(* CODESYS project Core.library
   Version: 1.3.3
   Title: Core
   DefaultNamespace: Core
   Placeholder: Core
   Company: Beckhoff Automation LLC

Project tree, tasks and I/O mapping:
  libraries: Tc2_Standard, * (Beckhoff Automation GmbH); Tc2_System, * (Beckhoff Automation GmbH); Tc3_DynamicMemory, * (Beckhoff Automation GmbH); Tc3_EventLogger, * (Beckhoff Automation GmbH); Tc3_JsonXml, * (Beckhoff Automation GmbH); Tc3_Module, * (Beckhoff Automation GmbH); Tc3_PackML_V3, * (Beckhoff Automation GmbH)
  _Interface/
    interface I_Base
    interface I_Command: Execute
    interface I_Disposable: Dispose
    interface I_Enablable: Disable, Enable, Enabled
    interface I_Initializable: Initialize, Initialized
    interface I_Override: Override
    interface I_Resettable: Reset
    interface I_Simulatable: Simulated
    interface I_Stoppable: Stop, Stopped
    interface I_TaskResult: Busy, Error, ErrorId
    interface I_ToString: ToString
  _Internal/
    Collection/
      Interface/
        interface I_Collection: AddItem, Clear, Count, IsEmpty, RemoveItem
        interface I_Enumerator: Current, CurrentItem, MoveToNext, ResetIterator
      function block Collection [ST]: FillGaps, AddItem, Clear, Count, Current, CurrentItem, IsEmpty, MoveToNext, RemoveItem, ResetIterator
    CollectionPeeker/
      Interface/
        interface I_CollectionPeeker: CollectionName, FirstItem, LastItem, MoveDownOne, MoveUpOne, PageDown, PageUp, PeekAt, Refresh
        interface I_Peekable: AcceptPeeker
        interface I_Peeker: PeekCollection
      function block CollectionPeeker [ST]: RefreshItems, UpdateEndItem, UpdateFirstItem, CollectionName, FirstItem, Items, LastItem, MoveDownOne, MoveUpOne, PageDown, PageUp, PeekAt, PeekCollection, Refresh
    Component/
      Interface/
        interface I_ComponentCollection: Accept, Count, GetAtIndex, GetComponentByName
        interface I_ContainComponents: Components, DeregisterComponent, DeregisterCyclic, DeregisterInitialize, RegisterComponent, RegisterCyclic, RegisterInitialize
      function block ComponentCollection [ST]: Accept, AddComponent, Count, GetAtIndex, GetComponentByName, RemoveComponent
    Cyclic/
      Interface/
        interface I_Cyclic: CyclicLogic
      function block CyclicRunner [ST]: AddCallee, CallAll, RemoveCallee
    Events/
      function block TcEventClassArguments [ST]: AddString, Clear, Event
    Initialize/
      function block Initializer [ST]: AddInitialize, Initialized, Initializing, RemoveInitialize
    List/
      Interface/
        interface I_List: ContainsItem, GetAtIndex, InsertAtIndex, RemoveAtIndex
      function block List [ST]: AddItem, Clear, RemoveItem, CountListItems, ContainsItem, Count, GetAtIndex, InsertAtIndex, RemoveAtIndex
    Module/
      Interface/
        interface I_ContainModules: DeregisterCyclic, DeregisterInitialize, DeregisterModule, Modules, RegisterCyclic, RegisterInitialize, RegisterModule
        interface I_ModuleCollection: Accept, Count, GetAtIndex, GetModuleByName
      function block ModuleCollection [ST]: Accept, AddModule, Count, GetAtIndex, GetModuleByName, RemoveModule
    Null/
      function block NullComponent [ST]
      function block NullItem [ST]
      function block NullModule [ST]: Accept, Components, DeregisterComponent, DeregisterCyclic, DeregisterInitialize, DeregisterModule, DeregisterWithParent, FB_Init, Modules, Name, RegisterComponent, RegisterCyclic, RegisterInitialize, RegisterModule, RegisterWithParent, ResetComponents, ResetModules
    Statemachine/
      Interface/
        interface I_StateList: AddStateAtIndex, GetStateAtIndex, NumberOfStates
      function block StateList [ST]: AddStateAtIndex, GetStateAtIndex, NumberOfStates
    Tracing/
      Interface/
        interface I_ContainTraceArgument: Arguments
        interface I_ContainTracePublisher: Publisher
        interface I_TraceArgument
        interface I_TraceInstanceLogger: LogMessageInstance
        interface I_TraceLogger: LogMessage
        interface I_TraceMessageInfo: Message, MessageId, Severity
        interface I_TracePublisher: Subscribe, Unsubscribe
        interface I_TraceSourceInfo: SourceId, SourceName, TimeStamp
      function block AdsLogger [ST]: FB_Init, LogMessage
      function block TcEventLogger [ST]: FB_Init, LogMessage
      function block TraceMessageInfo [ST]: Message, MessageId, Severity
      function block TraceSourceInfo [ST]: SourceId, SourceName, TimeStamp
      function USINT_To_TcEventSeverity [ST]
    Types/
      data type RegistrationResult
  Component/
    Interface/
      interface I_Component: Accept, DeregisterWithParent, Name, RegisterWithParent
      interface I_ComponentVisitor: VisitComponent
    function block Component [ST]: Accept, DeregisterWithParent, Name, RegisterWithParent, FB_Init
    function block CyclicComponent [ST]: CyclicLogic, DeregisterWithParent, RegisterWithParent
  Events/
    Interface/
      interface I_EventArguments: AddString, Clear
      interface I_EventClass: Arguments, ClearEventById, IsResettable, RaiseEvent, ResetBySeverity, SetEvent
      interface I_EventClassTcEvents: GenerateTcEvents, GetHighestActiveEventSeverity
      interface I_EventReaction: GetHighestActiveEventReaction, SetEventReactions
      interface I_EventReactionTcEvents: GetHighestActiveEventSeverity
    function block TcEventClass [ST]: Dispose, FB_Exit, ClearEventById, GetHighestActiveEventReaction, GetHighestActiveEventSeverity, IsResettable, RaiseEvent, ResetBySeverity, SetEvent, SetEventReactions, CheckEventId, FindActiveSeverity, GetEventAutoResetInstance, GetEventInstance, GetEventTriggerInstance, SetEventTriggerInstance, Reset, Arguments, CyclicLogic, GenerateTcEvents
  HMI/
    DUT/
      data type ST_HmiFunction
    Interface/
      interface I_Button: Active, Name, Permissive
      interface I_HmiFunction: ControlType, Disable, Enable, Enabled, InstancePath, LinkObject
      interface I_Permissive: OK, Set
      interface I_StringCollection: AddString, Clear, Entries
    function block Button [ST]: Active, Name, Permissive
    function block HmiFunction [ST]: ControlObject, ControlType, CyclicLogic, Disable, Enable, Enabled, InstancePath, LinkObject
  Modes/
    Interface/
      interface I_Mode: ChangeMode, CurrentMode
    function block ModeControl [ST]: ChangeMode, CurrentMode
    function block PackMLModeControl [ST]: ChangeMode, CurrentMode, CyclicLogic, StateMachine
  Module/
    Interface/
      interface I_Module: Accept, DeregisterWithParent, Name, RegisterWithParent, ResetComponents, ResetModules
      interface I_ModuleVisitor: VisitModule
    function block Module [ST]: FB_Init, CyclicLogic, OnCyclicCall, DeregisterComponent, DeregisterCyclic, DeregisterInitialize, DeregisterModule, DeregisterWithParent, Initialize, Initialized, Initializing, RegisterComponent, RegisterCyclic, RegisterInitialize, RegisterModule, RegisterWithParent, ResetComponents, ResetModules, Accept, Components, Modules, Name
  Module PackML/
    function block PackMLModule [ST]: FB_Init, Aborted, Aborting, Clearing, Completed, Completing, Execute, Held, Holding, Idle, Resetting, Starting, Stopped, Stopping, Suspended, Suspending, Unholding, Unsuspending, CyclicLogic, Statemachine, StateSelect
  Permissive Interlock/
    function block PermissiveInterlock [ST]: Check, OK, Set
  Project Information/
    function F_GetCompany [ST]
    function F_GetTitle [ST]
    function F_GetVersion [ST]
  Statemachine/
    DUT/
      data type ST_PackMLStatemachine_HMI
      data type ST_Statemachine_HMI
    Generic/
      function NextMinorStep [ST]
      function NextStep [ST]
      function SetStep [ST]
      function block State [ST]: Executing, FB_Init, Inactive
      function block Statemachine [ST]: Mode, ChangeState, CurrentState, States, CyclicLogic
      function block Statemachine_HMI [ST]: ControlObject, CyclicLogic, FB_Init
    Interface/
      interface I_ContainStatemachine: Statemachine
      interface I_State: Executing, Inactive
      interface I_Statemachine: ChangeState, CurrentState, Mode, States
    PackML/
      function block NextAvailablePackMLCommands [ST]: GetCommands
      function block PackMLStatemachine [ST]: Mode, CallState, ChangeState, CurrentState, States, CyclicLogic
      function block PackMLStatemachine_HMI [ST]: ControlObject, CyclicLogic, FB_Init
      function block PackMLStatemachine_ModuleIntegrated [ST]: Mode, ChangeState, CurrentState, CyclicLogic, StateComplete, States
  Tracing/
    DUT/
      data type TcEventSeverityExt
    Interface/
      interface I_Trace: Critical, Error, Info, Verbose, Warning
    global variables CoreTrace
    function block Trace [ST]: Critical, Error, Info, LogMessage, Subscribe, TraceLevel, Unsubscribe, Verbose, Warning
  Version/
    global variables Global_Version
  Visitors/
    Enable/
      function block CheckComponentsEnabledVisitor [ST]: Check, Enabled, VisitComponent
      function block DisableAllComponentsVisitor [ST]: Disable, Enabled, VisitComponent
      function block EnableAllComponentsVisitor [ST]: Enable, Enabled, VisitComponent
    Events/
      function block GetActiveEventSeverityVisitor [ST]: ActiveEventSeverity, FB_Init, VisitComponent, VisitModule
    HMI/
      function block GetSystemTreeJsonHmiVisitor [ST]: Clear, FB_Init, GetTree, VisitComponent, VisitModule
      function block HmiEnableDisableAllVisitor [ST]: DisableHmi, EnableHmi, VisitComponent, VisitModule
    Override/
      function block SetAllOverrideVisitor [ST]: Set, VisitComponent, VisitModule
    PackML Statemachine/
      function block ChangePackMLStateOnAllSubModulesVisitor [ST]: ChangeState, VisitModule
      function block EventReactorPackMLVisitor [ST]: CyclicLogic, FB_Init, VisitComponent, VisitModule
    Reset/
      function block GetComponentsTaskResultVisitor [ST]: Busy, Error, ErrorId, Update, VisitComponent
      function block ResetAllVisitor [ST]: Busy, Error, ErrorId, Reset, VisitComponent, VisitModule
      function block ResetComponentsVisitor [ST]: Busy, Error, ErrorId, Reset, VisitComponent
      function block ResetModulesVisitor [ST]: Busy, Error, ErrorId, Reset, VisitModule
    Statemachine/
      function block ChangeModeOnAllSubModulesVisitor [ST]: ChangeMode, VisitModule
      function block ChangeStateOnAllSubModulesVisitor [ST]: ChangeState, VisitModule
      function block EventReactorVisitor [ST]: CyclicLogic, FB_Init, VisitComponent, VisitModule
    Stop/
      function block StopAllComponentsVisitor [ST]: Stop, Stopped, VisitComponent
  global variables CoreParameter
  global variables GlobalCore
*)

// _Internal/Types/RegistrationResult
{attribute 'qualified_only'}
{attribute 'strict'}
{attribute 'to_string'}
TYPE RegistrationResult :
(
	Succeeded := 0,
	NullReference := -1,
	TooManyComponents := -2,
	AlreadyAdded := -3,
	CollectionEmpty := -4,
	NotFoundInCollection := -5
);
END_TYPE

// HMI/DUT/ST_HmiFunction
TYPE ST_HmiFunction :
	STRUCT
		Name	   : STRING;
		HmiEnabled : BOOL := TRUE;
	END_STRUCT
END_TYPE

// Statemachine/DUT/ST_PackMLStatemachine_HMI
TYPE ST_PackMLStatemachine_HMI EXTENDS ST_HmiFunction :
	STRUCT
		// Simplified Control
		ResetPermissive : BOOL;
		ResetPressed	: BOOL;
		Resetted		: BOOL;
		StartPermissive : BOOL;
		StartPressed	: BOOL;
		Started			: BOOL;
		StopPermissive	: BOOL;
		StopPressed		: BOOL;
		Stopped			: BOOL;
		// Standard Control
		CurrentMode	 : DINT;
		ModeCommand	 : DINT;
		CurrentState : E_PMLState;
		StateCommand : E_PMLCommand;
		// Next Available Commands
		NextAvailableCommands : ARRAY[0..9] OF E_PMLCommand;
	END_STRUCT
END_TYPE

// Statemachine/DUT/ST_Statemachine_HMI
TYPE ST_Statemachine_HMI EXTENDS ST_HmiFunction :
	STRUCT
		CurrentState	   : DINT;
		CurrentMode		   : DINT;
		StateChangeCommand : DINT;
		ModeChangeCommand  : DINT;
	END_STRUCT
END_TYPE

// Tracing/DUT/TcEventSeverityExt
{attribute 'qualified_only'}
{attribute 'strict'}
{attribute 'to_string'}
TYPE TcEventSeverityExt : (
		Verbose	 := 0,
		Info	 := 1,
		Warning	 := 2,
		Error	 := 3,
		Critical := 4,
		Off		 := 5
	);
END_TYPE

// Tracing/CoreTrace
VAR_GLOBAL
	Trace : Trace<CoreParameter.MaxCountInCollections> := (TraceLevel := CoreParameter.TraceLevel);
	{attribute 'hide'}
	TcEventLogger : TcEventLogger(Trace);
	{attribute 'hide'}
	AdsLogger : AdsLogger(Trace);
END_VAR

// Version/Global_Version
{attribute 'TcGenerated'}
{attribute 'no-analysis'}
{attribute 'linkalways'}
// This function has been automatically generated from the project information.
VAR_GLOBAL CONSTANT
	{attribute 'const_non_replaced'}
	stLibVersion_Core : ST_LibVersion := (iMajor := 1, iMinor := 3, iBuild := 3, iRevision := 0, nFlags := 0, sVersion := '1.3.3');
END_VAR

// CoreParameter
{attribute 'qualified_only'}
VAR_GLOBAL CONSTANT
	MaxCountInCollections : UDINT			   := 50;
	EnableTcEventLogging  : BOOL			   := FALSE;
	EnableAdsLogger		  : BOOL			   := TRUE;
	ClearingTimeout		  : TIME			   := T#2S;
	TraceLevel			  : TcEventSeverityExt := TcEventSeverityExt.Verbose;
END_VAR

// GlobalCore
{attribute 'qualified_only'}
VAR_GLOBAL
	DynamicMemory : FB_DynMem_Manager;
END_VAR

// _Interface/I_Base
INTERFACE I_Base EXTENDS __SYSTEM.IQueryInterface

END_INTERFACE

// _Interface/I_Command
INTERFACE I_Command EXTENDS I_Base

METHOD Execute : BOOL
VAR_INPUT
END_VAR
END_METHOD

END_INTERFACE

// _Interface/I_Disposable
INTERFACE I_Disposable EXTENDS I_Base

METHOD Dispose
VAR_INPUT
END_VAR
END_METHOD

END_INTERFACE

// _Interface/I_Enablable
INTERFACE I_Enablable EXTENDS I_Base

METHOD Disable
VAR_INPUT
END_VAR
END_METHOD

METHOD Enable
VAR_INPUT
END_VAR
END_METHOD

{attribute 'monitoring' := 'call'}
PROPERTY Enabled : BOOL
GET
END_GET
END_PROPERTY

END_INTERFACE

// _Interface/I_Initializable
INTERFACE I_Initializable EXTENDS I_Base

METHOD Initialize
END_METHOD

{attribute 'monitoring' := 'call'}
PROPERTY Initialized : BOOL
GET
END_GET
SET
END_SET
END_PROPERTY

END_INTERFACE

// _Interface/I_Override
INTERFACE I_Override EXTENDS I_Base

{attribute 'monitoring' := 'call'}
PROPERTY Override : LREAL
SET
END_SET
END_PROPERTY

END_INTERFACE

// _Interface/I_Resettable
INTERFACE I_Resettable EXTENDS I_Base

METHOD Reset
END_METHOD

END_INTERFACE

// _Interface/I_Simulatable
INTERFACE I_Simulatable EXTENDS I_Base

{attribute 'monitoring' := 'call'}
PROPERTY Simulated : BOOL
GET
END_GET
SET
END_SET
END_PROPERTY

END_INTERFACE

// _Interface/I_Stoppable
INTERFACE I_Stoppable EXTENDS I_Base

METHOD Stop
VAR_INPUT
END_VAR
END_METHOD

{attribute 'monitoring' := 'call'}
PROPERTY Stopped : BOOL
GET
END_GET
END_PROPERTY

END_INTERFACE

// _Interface/I_TaskResult
INTERFACE I_TaskResult EXTENDS I_Base

{attribute 'monitoring' := 'call'}
PROPERTY Busy : BOOL
GET
END_GET
END_PROPERTY

{attribute 'monitoring' := 'call'}
PROPERTY Error : BOOL
GET
END_GET
END_PROPERTY

{attribute 'monitoring' := 'call'}
PROPERTY ErrorId : UDINT
GET
END_GET
END_PROPERTY

END_INTERFACE

// _Interface/I_ToString
INTERFACE I_ToString EXTENDS I_Base

METHOD ToString : T_MaxString
VAR_INPUT
END_VAR
END_METHOD

END_INTERFACE

// _Internal/Collection/Interface/I_Collection
INTERFACE I_Collection EXTENDS I_Enumerator

METHOD AddItem
VAR_INPUT
	Item : I_Base;
END_VAR
END_METHOD

METHOD Clear
VAR_INPUT
END_VAR
END_METHOD

{attribute 'monitoring' := 'call'}
PROPERTY Count : UDINT
GET
END_GET
END_PROPERTY

{attribute 'monitoring' := 'call'}
PROPERTY IsEmpty : BOOL
GET
END_GET
END_PROPERTY

METHOD RemoveItem
VAR_INPUT
	Item : I_Base;
END_VAR
END_METHOD

END_INTERFACE

// _Internal/Collection/Interface/I_Enumerator
INTERFACE I_Enumerator

PROPERTY Current : I_Base
GET
END_GET
END_PROPERTY

{attribute 'monitoring' := 'call'}
PROPERTY CurrentItem : UDINT
GET
END_GET
END_PROPERTY

PROPERTY MoveToNext : BOOL
GET
END_GET
END_PROPERTY

METHOD ResetIterator
VAR_INPUT
END_VAR
END_METHOD

END_INTERFACE

// _Internal/Collection/Collection
FUNCTION_BLOCK Collection
VAR_GENERIC CONSTANT
	CollectionSize : UDINT := 1;
END_VAR IMPLEMENTS I_Collection, I_Enumerator
VAR
	{attribute 'instance-path'}
	{attribute 'noinit'}
	InstancePath  : STRING;
	_Data		  : ARRAY[0..CollectionSize - 1] OF I_Base;
	_Current	  : I_Base;
	_Count		  : UDINT;
	_CurrentIndex : UDINT;
	{attribute 'hide'}
	NullItem : NullItem;
	{attribute 'hide'}
	ipNullItem : I_Base := NullItem;
END_VAR

METHOD PROTECTED FillGaps
VAR
	Item	 : I_Base;
	ItemNext : I_Base;
	i		 : UDINT;
END_VAR
IF _Count > 1 THEN
	FOR i := 0 TO (_Count - 2) DO
		Item	 := _Data[i];
		ItemNext := _Data[i + 1];
		IF Item = 0 AND ItemNext <> 0 THEN
			_Data[i]	 := ItemNext;
			_Data[i + 1] := 0;
		END_IF
	END_FOR
END_IF
END_METHOD

METHOD AddItem
VAR_INPUT
	Item	: I_Base;
END_VAR
IF Item = 0 THEN
	Trace.Error(InstancePath, 'No Items to add to this Collection!');
	RETURN;
END_IF

IF _Count > CollectionSize - 1 THEN
	Trace.Error(InstancePath, 'No space left in Collection, increase size!');
	RETURN;
END_IF

_Data[_Count] := Item;
_Count		  := _Count + 1;
END_METHOD

METHOD Clear
VAR
	i : UDINT;
END_VAR
IF _Count = 0 THEN
	RETURN;
END_IF

FOR i := 0 TO _Count - 1 DO
	_Data[i] := 0;
END_FOR

_Count := 0;
ResetIterator();
END_METHOD

{attribute 'monitoring' := 'call'}
PROPERTY Count : UDINT
GET
Count := _Count;
END_GET
END_PROPERTY

PROPERTY Current : I_Base
GET
IF _Current <> 0 THEN
	Current := _Current; 
END_IF
END_GET
END_PROPERTY

{attribute 'monitoring' := 'call'}
PROPERTY CurrentItem : UDINT
GET
CurrentItem := _CurrentIndex;
END_GET
END_PROPERTY

{attribute 'monitoring' := 'call'}
PROPERTY IsEmpty : BOOL
GET
IsEmpty := _Count = 0;
END_GET
END_PROPERTY

PROPERTY MoveToNext : BOOL
GET
MoveToNext := FALSE;
IF Count = 0 THEN
	RETURN;
END_IF

IF _CurrentIndex = Count THEN
	RETURN;
END_IF

_Current	  := _Data[_CurrentIndex];
_CurrentIndex := _CurrentIndex + 1;
MoveToNext	  := TRUE;
END_GET
END_PROPERTY

METHOD RemoveItem
VAR_INPUT
	Item : I_Base;
END_VAR

VAR
	i		  : UDINT;
	ItemFound : BOOL;
END_VAR
IF _Count = 0 THEN
	Trace.LogMessage(InstancePath, 'No Items found in this Collection!');
	RETURN;
END_IF

IF Item = 0 THEN
	Trace.LogMessage(InstancePath, 'Item to remove needs to be valid interface!');
	RETURN;
END_IF

FOR i := 0 TO (_Count - 1) DO
	IF _Data[i] = Item THEN
		_Data[i]  := 0;
		ItemFound := TRUE;
	END_IF
END_FOR

FillGaps();
IF ItemFound THEN
	_Count := _Count - 1;
END_IF
END_METHOD

METHOD ResetIterator
_Current	  := ipNullItem;
_CurrentIndex := 0;
END_METHOD

END_FUNCTION_BLOCK

// _Internal/Null/NullItem
FUNCTION_BLOCK NullItem IMPLEMENTS I_Base
VAR
END_VAR

END_FUNCTION_BLOCK

// Tracing/Trace
FUNCTION_BLOCK Trace
VAR_GENERIC CONSTANT
	MaxCount : UDINT := 10;
END_VAR IMPLEMENTS I_TracePublisher, I_Trace
VAR
	Loggers : ARRAY[0..MaxCount] OF I_TraceLogger;
	_TraceLevel : TcEventSeverityExt := TcEventSeverityExt.Warning;
END_VAR

METHOD Critical
VAR_INPUT
	Source	  : T_MaxString;
	Message	  : T_MaxString;
END_VAR
VAR
	i : UDINT;
END_VAR
FOR i := 0 TO MaxCount DO
	IF Loggers[i] <> 0 AND_THEN _TraceLevel < 5 THEN
		Loggers[i].LogMessage(Source,
							  Message,
							  0,
							  0,
							  1,
							  4);
	END_IF
END_FOR
END_METHOD

METHOD Error
VAR_INPUT
	Source	  : T_MaxString;
	Message	  : T_MaxString;
END_VAR
VAR
	i : UDINT;
END_VAR
FOR i := 0 TO MaxCount DO
	IF Loggers[i] <> 0 AND_THEN _TraceLevel < 4 THEN
		Loggers[i].LogMessage(Source,
							  Message,
							  0,
							  0,
							  1,
							  3);
	END_IF
END_FOR
END_METHOD

METHOD Info
VAR_INPUT
	Source	  : T_MaxString;
	Message	  : T_MaxString;
END_VAR
VAR
	i : UDINT;
END_VAR
FOR i := 0 TO MaxCount DO
	IF Loggers[i] <> 0 AND_THEN _TraceLevel < 2 THEN
		Loggers[i].LogMessage(Source,
							  Message,
							  0,
							  0,
							  1,
							  1);
	END_IF
END_FOR
END_METHOD

METHOD LogMessage
VAR_INPUT
	Key		  : T_MaxString;
	Value	  : T_MaxString;
	SourceId  : UDINT := 0;
	TimeStamp : ULINT := 0;
	MessageId : UDINT := 1;
	Severity  : USINT := 1;
END_VAR

VAR
	i : UDINT;
END_VAR
FOR i := 0 TO MaxCount DO
	IF Loggers[i] <> 0 THEN
		Loggers[i].LogMessage(Key,
							  Value,
							  SourceId,
							  TimeStamp,
							  MessageId,
							  Severity);
	END_IF
END_FOR
END_METHOD

METHOD Subscribe
VAR_INPUT
	Logger : I_TraceLogger;
END_VAR

VAR
	i : UDINT;
END_VAR
FOR i := 0 TO CoreParameter.MaxCountInCollections DO
	IF Loggers[i] = 0 THEN
		Loggers[i] := Logger;
		EXIT;
	END_IF
END_FOR
END_METHOD

PROPERTY TraceLevel : TcEventSeverityExt
GET
TraceLevel := _TraceLevel;
END_GET
SET
_TraceLevel := TraceLevel;
END_SET
END_PROPERTY

METHOD Unsubscribe
VAR_INPUT
	Logger : I_TraceLogger;
END_VAR

VAR
	i : UDINT;
END_VAR
FOR i := 0 TO CoreParameter.MaxCountInCollections DO
	IF Loggers[i] = Logger THEN
		Loggers[i] := 0;
		EXIT;
	END_IF
END_FOR
END_METHOD

METHOD Verbose
VAR_INPUT
	Source	  : T_MaxString;
	Message	  : T_MaxString;
END_VAR
VAR
	i : UDINT;
END_VAR
FOR i := 0 TO MaxCount DO
	IF Loggers[i] <> 0 AND_THEN _TraceLevel = 0 THEN
		Loggers[i].LogMessage(Source,
							  Message,
							  0,
							  0,
							  1,
							  0);
	END_IF
END_FOR
END_METHOD

METHOD Warning
VAR_INPUT
	Source	  : T_MaxString;
	Message	  : T_MaxString;
END_VAR
VAR
	i : UDINT;
END_VAR
FOR i := 0 TO MaxCount DO
	IF Loggers[i] <> 0 AND_THEN _TraceLevel < 3 THEN
		Loggers[i].LogMessage(Source,
							  Message,
							  0,
							  0,
							  1,
							  2);
	END_IF
END_FOR
END_METHOD

END_FUNCTION_BLOCK

// _Internal/Tracing/Interface/I_TracePublisher
INTERFACE I_TracePublisher

METHOD Subscribe
VAR_INPUT
	Logger : I_TraceLogger;
END_VAR
END_METHOD

METHOD Unsubscribe
VAR_INPUT
	Logger : I_TraceLogger;
END_VAR
END_METHOD

END_INTERFACE

// _Internal/Tracing/Interface/I_TraceLogger
INTERFACE I_TraceLogger EXTENDS I_Base

METHOD LogMessage
VAR_INPUT
	Key		  : T_MaxString;
	Value	  : T_MaxString;
	SourceId  : UDINT := 0;
	TimeStamp : ULINT := 0;
	MessageId : UDINT := 1;
	Severity  : USINT := 1;
END_VAR
END_METHOD

END_INTERFACE

// Tracing/Interface/I_Trace
INTERFACE I_Trace

METHOD Critical
VAR_INPUT
	Source	  : T_MaxString;
	Message	  : T_MaxString;
END_VAR
END_METHOD

METHOD Error
VAR_INPUT
	Source	  : T_MaxString;
	Message	  : T_MaxString;
END_VAR
END_METHOD

METHOD Info
VAR_INPUT
	Source	  : T_MaxString;
	Message	  : T_MaxString;
END_VAR
END_METHOD

METHOD Verbose
VAR_INPUT
	Source	  : T_MaxString;
	Message	  : T_MaxString;
END_VAR
END_METHOD

METHOD Warning
VAR_INPUT
	Source	  : T_MaxString;
	Message	  : T_MaxString;
END_VAR
END_METHOD

END_INTERFACE

// _Internal/CollectionPeeker/Interface/I_CollectionPeeker
INTERFACE I_CollectionPeeker EXTENDS I_Base

{attribute 'monitoring':='call'}
PROPERTY CollectionName : T_MaxString
GET
END_GET
SET
END_SET
END_PROPERTY

{attribute 'monitoring':='call'}
PROPERTY FirstItem : UDINT
GET
END_GET
END_PROPERTY

{attribute 'monitoring':='call'}
PROPERTY LastItem : UDINT
GET
END_GET
END_PROPERTY

{attribute 'monitoring' := 'call'}
PROPERTY MoveDownOne : BOOL
SET
END_SET
END_PROPERTY

{attribute 'monitoring' := 'call'}
PROPERTY MoveUpOne : BOOL
SET
END_SET
END_PROPERTY

{attribute 'monitoring' := 'call'}
PROPERTY PageDown : BOOL
SET
END_SET
END_PROPERTY

{attribute 'monitoring' := 'call'}
PROPERTY PageUp : BOOL
SET
END_SET
END_PROPERTY

METHOD PeekAt
VAR_INPUT
	Peekable : I_Peekable;
END_VAR
END_METHOD

{attribute 'monitoring':='call'}
PROPERTY Refresh : BOOL
GET
END_GET
SET
END_SET
END_PROPERTY

END_INTERFACE

// _Internal/CollectionPeeker/Interface/I_Peekable
INTERFACE I_Peekable EXTENDS I_Base

METHOD AcceptPeeker
VAR_INPUT
	Peeker : I_Peeker;
END_VAR
END_METHOD

END_INTERFACE

// _Internal/CollectionPeeker/Interface/I_Peeker
INTERFACE I_Peeker EXTENDS I_Base

METHOD PeekCollection
VAR_INPUT
	Collection : I_Collection;
END_VAR
END_METHOD

END_INTERFACE

// _Internal/CollectionPeeker/CollectionPeeker
{attribute 'hide_all_locals'}
FUNCTION_BLOCK CollectionPeeker
VAR_GENERIC CONSTANT
	Peek_Size : UDINT := 5;
END_VAR IMPLEMENTS I_CollectionPeeker, I_Peeker
VAR
	_CurrentItem	: UDINT;
	_EndItem		: UDINT;
	_CollectionName : T_MaxString;
	_Collection		: I_Collection;
	_Items			: ARRAY[1..Peek_Size] OF I_Base;
END_VAR

METHOD PRIVATE RefreshItems
VAR
	startItem  : UDINT;
	endItem	   : UDINT;
	i		   : UDINT := 1;
	wrapAround : BOOL;
END_VAR
MEMSET(ADR(_Items), 0, SIZEOF(_Items));
IF _CurrentItem > _EndItem THEN //we're wrapped around
	i		   := 1 + ((_Collection.Count - _CurrentItem) + 1);
	wrapAround := TRUE;
END_IF

_Collection.ResetIterator();
WHILE _Collection.MoveToNext DO
	IF _Collection.CurrentItem >= _CurrentItem AND _Collection.CurrentItem <= _EndItem THEN
		_Items[i] := _Collection.Current;
		i		  := i + 1;
	ELSIF wrapAround AND (_Collection.CurrentItem >= _CurrentItem OR _Collection.CurrentItem <= _EndItem) THEN
		_Items[i] := _Collection.Current;
		i		  := i + 1;
		IF i > Peek_Size THEN
			i := 1;
		END_IF
	END_IF
END_WHILE
END_METHOD

METHOD PRIVATE UpdateEndItem
VAR_INPUT
END_VAR
_EndItem := _CurrentItem + Peek_Size - 1;
IF _EndItem > _Collection.Count THEN
	_EndItem := _EndItem - _Collection.Count;
END_IF
END_METHOD

METHOD PRIVATE UpdateFirstItem
VAR_INPUT
END_VAR
END_METHOD

{attribute 'monitoring':='call'}
PROPERTY CollectionName : T_MaxString
GET
CollectionName := _CollectionName;
END_GET
SET
_CollectionName := CollectionName;
END_SET
END_PROPERTY

{attribute 'monitoring' := 'call'}
PROPERTY FirstItem : UDINT
GET
FirstItem := _CurrentItem;
END_GET
SET
IF _Collection = 0 THEN
	RETURN;
END_IF

IF FirstItem > _Collection.Count OR FirstItem < 1 THEN
	RETURN;
END_IF

_CurrentItem := FirstItem;
UpdateEndItem();
RefreshItems();
END_SET
END_PROPERTY

{attribute 'monitoring' := 'call'}
PROPERTY Items : REFERENCE TO ARRAY[1..Peek_Size] OF I_Base
GET
Items REF= _Items;
END_GET
END_PROPERTY

{attribute 'monitoring' := 'call'}
PROPERTY LastItem : UDINT
GET
LastItem := _EndItem;
END_GET
END_PROPERTY

{attribute 'monitoring' := 'call'}
PROPERTY MoveDownOne : BOOL
GET
END_GET
SET
IF _Collection = 0 OR NOT MoveDownOne THEN
	RETURN;
END_IF

IF _Collection.Count <= Peek_Size THEN
	RETURN;
END_IF

_CurrentItem := _CurrentItem + 1;
IF _CurrentItem > _Collection.Count THEN
	_CurrentItem := 1;
END_IF

UpdateEndItem();
RefreshItems();
END_SET
END_PROPERTY

{attribute 'monitoring' := 'call'}
PROPERTY MoveUpOne : BOOL
GET
END_GET
SET
IF _Collection = 0 THEN
	RETURN;
END_IF

IF _Collection.Count <= Peek_Size THEN
	RETURN;
END_IF

_CurrentItem := _CurrentItem - 1;
IF _CurrentItem < 1 THEN
	_CurrentItem := _Collection.Count;
END_IF

UpdateEndItem();
RefreshItems();
END_SET
END_PROPERTY

{attribute 'monitoring' := 'call'}
PROPERTY PageDown : BOOL
GET
END_GET
SET
IF _Collection = 0 OR NOT PageDown THEN
	RETURN;
END_IF

IF _Collection.Count <= Peek_Size THEN
	RETURN;
END_IF

IF _CurrentItem > (_Collection.Count - Peek_Size) THEN
	_CurrentItem := (Peek_Size - (_Collection.Count - _CurrentItem));
ELSE
	_CurrentItem := _CurrentItem + Peek_Size;
END_IF

UpdateEndItem();
RefreshItems();
END_SET
END_PROPERTY

{attribute 'monitoring' := 'call'}
PROPERTY PageUp : BOOL
GET
END_GET
SET
VAR
	tmp : UDINT;
END_VAR
IF _Collection = 0 OR NOT PageUp THEN
	RETURN;
END_IF

IF _Collection.Count <= Peek_Size THEN
	RETURN;
END_IF

IF _CurrentItem < Peek_Size THEN
	_CurrentItem := (_Collection.Count - (Peek_Size - _CurrentItem));
ELSE
	_CurrentItem := _CurrentItem - Peek_Size;
END_IF

UpdateEndItem();
RefreshItems();
END_SET
END_PROPERTY

METHOD PeekAt
VAR_INPUT
	Peekable : I_Peekable;
END_VAR
Peekable.AcceptPeeker(THIS^);
END_METHOD

METHOD PeekCollection
VAR_INPUT
	Collection : I_Collection;
END_VAR
_Collection	 := Collection;
_CurrentItem := 1;
_EndItem	 := Peek_Size;
RefreshItems();
END_METHOD

{attribute 'monitoring':='call'}
PROPERTY Refresh : BOOL
GET
END_GET
SET
IF _Collection <> 0 AND Refresh THEN
	RefreshItems();
END_IF
END_SET
END_PROPERTY

END_FUNCTION_BLOCK

// _Internal/Component/Interface/I_ComponentCollection
INTERFACE I_ComponentCollection

METHOD Accept
VAR_INPUT
	Visitor : I_ComponentVisitor;
END_VAR
END_METHOD

{attribute 'monitoring' := 'call'}
PROPERTY Count : UDINT
GET
END_GET
END_PROPERTY

METHOD GetAtIndex : I_Component
VAR_INPUT
	Index : UDINT;
END_VAR
END_METHOD

METHOD GetComponentByName : I_Component
VAR_INPUT
	Name : T_MaxString;
END_VAR
END_METHOD

END_INTERFACE

// Component/Interface/I_ComponentVisitor
INTERFACE I_ComponentVisitor

METHOD VisitComponent
VAR_INPUT
	Component : I_Component;
END_VAR
END_METHOD

END_INTERFACE

// Component/Component
FUNCTION_BLOCK ABSTRACT Component IMPLEMENTS I_Component
VAR
	_Name : T_MaxString;
	RegisteredAsComponentResult : RegistrationResult;
END_VAR

METHOD Accept
VAR_INPUT
	ComponentVisitor : I_ComponentVisitor;
END_VAR
ComponentVisitor.VisitComponent(THIS^);
END_METHOD

METHOD DeregisterWithParent
VAR_INPUT
	Parent : I_ContainComponents;
END_VAR
Parent.DeregisterComponent(THIS^);
END_METHOD

{attribute 'monitoring' := 'call'}
PROPERTY Name : T_MaxString
GET
Name := _Name;
END_GET
SET
_Name := Name;
END_SET
END_PROPERTY

METHOD RegisterWithParent
VAR_INPUT
	Parent : I_ContainComponents;
END_VAR
RegisteredAsComponentResult := Parent.RegisterComponent(THIS^);
END_METHOD

//FB_Init is always available implicitly and it is used primarily for initialization.

//The return value is not evaluated. For a specific influence, you can also declare the

//methods explicitly and provide additional code there with the standard initialization

//code. You can evaluate the return value.
METHOD FB_Init : BOOL
VAR_INPUT
	bInitRetains : BOOL; // TRUE: the retain variables are initialized (reset warm / reset cold)
	bInCopyCode	 : BOOL; // TRUE: the instance will be copied to the copy code afterward (online change)   
	Name		 : T_MaxString;
END_VAR
_Name := Name;
END_METHOD

END_FUNCTION_BLOCK

// Component/Interface/I_Component
INTERFACE I_Component EXTENDS I_Base

METHOD Accept
VAR_INPUT
	ComponentVisitor : I_ComponentVisitor;
END_VAR
END_METHOD

METHOD DeregisterWithParent
VAR_INPUT
	Parent : I_ContainComponents;
END_VAR
END_METHOD

{attribute 'monitoring' := 'call'}
PROPERTY Name : T_MaxString
GET
END_GET
SET
END_SET
END_PROPERTY

METHOD RegisterWithParent
VAR_INPUT
	Parent : I_ContainComponents;
END_VAR
END_METHOD

END_INTERFACE

// _Internal/Component/Interface/I_ContainComponents
INTERFACE I_ContainComponents

PROPERTY Components : I_ComponentCollection
GET
END_GET
END_PROPERTY

METHOD DeregisterComponent  : RegistrationResult
VAR_INPUT
	Component : I_Component;
END_VAR
END_METHOD

METHOD DeregisterCyclic : RegistrationResult
VAR_INPUT
	Cyclic : I_Cyclic;
END_VAR
END_METHOD

METHOD DeregisterInitialize : RegistrationResult
VAR_INPUT
	Initializable : I_Initializable;
END_VAR
END_METHOD

METHOD RegisterComponent  : RegistrationResult
VAR_INPUT
	Component : I_Component;
END_VAR
END_METHOD

METHOD RegisterCyclic  : RegistrationResult
VAR_INPUT
	Cyclic : I_Cyclic;
END_VAR
END_METHOD

METHOD RegisterInitialize  : RegistrationResult
VAR_INPUT
	Initializable : I_Initializable;
END_VAR
END_METHOD

END_INTERFACE

// _Internal/Cyclic/Interface/I_Cyclic
INTERFACE I_Cyclic EXTENDS I_Base

METHOD CyclicLogic
VAR_INPUT
END_VAR
END_METHOD

END_INTERFACE

// _Internal/Component/ComponentCollection
FUNCTION_BLOCK ComponentCollection
VAR_GENERIC CONSTANT
	MaxCount : UDINT := 10;
END_VAR IMPLEMENTS I_ComponentCollection
VAR
	Components	   : ARRAY[0..MaxCount] OF I_Component;
	ComponentCount : UDINT;
	NullComponent  : NullComponent('Null Component');
END_VAR

METHOD Accept
VAR_INPUT
	Visitor : I_ComponentVisitor;
END_VAR

VAR
	i : UDINT;
END_VAR
FOR i := 0 TO MaxCount DO
	IF Components[i] = 0 THEN
		EXIT;
	END_IF

	Components[i].Accept(Visitor);
END_FOR
END_METHOD

METHOD AddComponent : RegistrationResult
VAR_INPUT
	Component : I_Component;
END_VAR

VAR
	i : UDINT;
	Registered : BOOL;
END_VAR
IF Component = 0 THEN
	AddComponent := RegistrationResult.NullReference;
	RETURN;
END_IF

IF ComponentCount >= MaxCount THEN
	AddComponent := RegistrationResult.TooManyComponents;
	RETURN;
END_IF

FOR i := 0 TO MaxCount DO
	IF Components[i] = Component THEN
		Registered := TRUE;
	END_IF
END_FOR

IF Registered THEN
	AddComponent := RegistrationResult.AlreadyAdded;
	RETURN;
END_IF

FOR i := 0 TO MaxCount DO
	IF Components[i] = 0 THEN
		Components[i] := Component;
		ComponentCount := ComponentCount + 1;
		EXIT;
	END_IF
END_FOR
END_METHOD

{attribute 'monitoring' := 'call'}
PROPERTY Count : UDINT
GET
Count := TO_UDINT(ComponentCount);
END_GET
END_PROPERTY

METHOD GetAtIndex : I_Component
VAR_INPUT
	Index : UDINT;
END_VAR
IF Index > Count THEN
	GetAtIndex := NullComponent;
	RETURN;
END_IF

IF Index < 0 THEN
	GetAtIndex := NullComponent;
	RETURN;
END_IF

IF Components[Index] <> 0 THEN
	GetAtIndex := Components[Index];
ELSE
	GetAtIndex := NullComponent;
END_IF
END_METHOD

METHOD GetComponentByName : I_Component
VAR_INPUT
	Name : T_MaxString;
END_VAR

VAR
	i : UDINT;
END_VAR
FOR i := 0 TO MaxCount DO
	IF Components[i] = 0 THEN
		EXIT;
	END_IF

	IF Components[i].Name = Name THEN
		GetComponentByName := Components[i];
		EXIT;
	END_IF
END_FOR
END_METHOD

METHOD RemoveComponent : RegistrationResult
VAR_INPUT
	Component : I_Component;
END_VAR

VAR
	i : UDINT;
	PresentInCollection : BOOL;
END_VAR
IF Component = 0 THEN
	RemoveComponent := RegistrationResult.NullReference;
	RETURN;
END_IF

IF ComponentCount = 0 THEN
	RemoveComponent := RegistrationResult.CollectionEmpty;
	RETURN;
END_IF

FOR i := 0 TO MaxCount DO
	IF Components[i] = Component THEN
		PresentInCollection := TRUE;
	END_IF
END_FOR

IF NOT PresentInCollection THEN
	RemoveComponent := RegistrationResult.NotFoundInCollection;
	RETURN;
END_IF

FOR i := 0 TO MaxCount DO
	IF Components[i] = Component THEN
		ComponentCount := ComponentCount - 1;
		IF i < MaxCount THEN
			MEMMOVE(ADR(Components[i]), ADR(Components[i + 1]), (MaxCount - i) * SIZEOF(Component));
		ELSE
			Components[MaxCount] := 0;
		END_IF
		EXIT;
	END_IF
END_FOR
END_METHOD

END_FUNCTION_BLOCK

// _Internal/Null/NullComponent
FUNCTION_BLOCK NullComponent EXTENDS Component
VAR
END_VAR

END_FUNCTION_BLOCK

// _Internal/Cyclic/CyclicRunner
FUNCTION_BLOCK CyclicRunner
VAR_GENERIC CONSTANT
	MaxCount : UDINT := 10;
END_VAR

VAR
	Callees		: ARRAY[0..MaxCount] OF I_Cyclic;
	CalleeCount : UDINT;
END_VAR

METHOD AddCallee : RegistrationResult
VAR_INPUT
	Callee : I_Cyclic;
END_VAR

VAR
	i : UDINT;
	Registered : BOOL;
END_VAR
IF Callee = 0 THEN
	AddCallee := RegistrationResult.NullReference;
	RETURN;
END_IF

IF CalleeCount >= MaxCount THEN
	AddCallee := RegistrationResult.TooManyComponents;
	RETURN;
END_IF

FOR i := 0 TO MaxCount DO
	IF Callees[i] = Callee THEN
		Registered := TRUE;
	END_IF
END_FOR

IF Registered THEN
	AddCallee := RegistrationResult.AlreadyAdded;
	RETURN;
END_IF

FOR i := 0 TO MaxCount DO
	IF Callees[i] = 0 THEN
		Callees[i] := Callee;
		CalleeCount := CalleeCount + 1;
		EXIT;
	END_IF
END_FOR
END_METHOD

METHOD CallAll
VAR_INST
	Logged : BOOL;
END_VAR

VAR
	i	   : UDINT;
	Callee : I_Cyclic;
END_VAR
FOR i := 0 TO MaxCount DO
	IF Callees[i] = 0 THEN
		RETURN;
	END_IF

	Callees[i].CyclicLogic();
END_FOR

IF NOT Logged THEN
	Logged := TRUE;
	Trace.LogMessage('Cyclic Runner', 'Collection is full. Review library parameters and code to ensure proper setup.');
END_IF
END_METHOD

METHOD RemoveCallee : RegistrationResult
VAR_INPUT
	Callee : I_Cyclic;
END_VAR

VAR
	i : UDINT;
	PresentInCollection : BOOL;
END_VAR
IF Callee = 0 THEN
	RemoveCallee := RegistrationResult.NullReference;
	RETURN;
END_IF

IF CalleeCount = 0 THEN
	RemoveCallee := RegistrationResult.CollectionEmpty;
	RETURN;
END_IF

FOR i := 0 TO MaxCount DO
	IF Callees[i] = Callee THEN
		PresentInCollection := TRUE;
	END_IF
END_FOR

IF NOT PresentInCollection THEN
	RemoveCallee := RegistrationResult.NotFoundInCollection;
	RETURN;
END_IF

FOR i := 0 TO MaxCount DO
	IF Callees[i] = Callee THEN
		CalleeCount := CalleeCount - 1;
		IF i < MaxCount THEN
			MEMMOVE(ADR(Callees[i]), ADR(Callees[i + 1]), (MaxCount - i) * SIZEOF(Callee));
		ELSE
			Callees[MaxCount] := 0;
		END_IF
		EXIT;
	END_IF
END_FOR
END_METHOD

END_FUNCTION_BLOCK

// _Internal/Events/TcEventClassArguments
FUNCTION_BLOCK TcEventClassArguments IMPLEMENTS I_EventArguments
VAR
	pArgumentEvent : POINTER TO FB_TcAlarm;
END_VAR

METHOD AddString : I_EventArguments
VAR_INPUT
	Argument : STRING;
END_VAR
IF pArgumentEvent <> 0 THEN
	pArgumentEvent^.ipArguments.AddString(Argument);
END_IF

AddString := THIS^;
END_METHOD

METHOD Clear : I_EventArguments
IF pArgumentEvent <> 0 THEN
	pArgumentEvent^.ipArguments.Clear();
END_IF

Clear := THIS^;
END_METHOD

PROPERTY Event : POINTER TO FB_TcAlarm
SET
pArgumentEvent := Event;
END_SET
END_PROPERTY

END_FUNCTION_BLOCK

// Events/Interface/I_EventArguments
INTERFACE I_EventArguments EXTENDS I_Base

METHOD AddString : I_EventArguments
VAR_INPUT
	Argument : STRING;
END_VAR
END_METHOD

METHOD Clear : I_EventArguments
VAR_INPUT
END_VAR
END_METHOD

END_INTERFACE

// _Internal/Initialize/Initializer
FUNCTION_BLOCK Initializer
VAR_GENERIC CONSTANT
	MaxCount : UDINT := 10;
END_VAR

VAR
	Initializable : ARRAY[0..MaxCount] OF I_Initializable;
	InitializableCount : UDINT;
END_VAR

METHOD AddInitialize : RegistrationResult
VAR_INPUT
	Initialize : I_Initializable;
END_VAR

VAR
	i : UDINT;
	Registered : BOOL;
END_VAR
IF Initialize = 0 THEN
	AddInitialize := RegistrationResult.NullReference;
	RETURN;
END_IF

IF InitializableCount >= MaxCount THEN
	AddInitialize := RegistrationResult.TooManyComponents;
	RETURN;
END_IF

FOR i := 0 TO MaxCount DO
	IF Initializable[i] = Initialize THEN
		Registered := TRUE;
	END_IF
END_FOR

IF Registered THEN
	AddInitialize := RegistrationResult.AlreadyAdded;
	RETURN;
END_IF

FOR i := 0 TO MaxCount DO
	IF Initializable[i] = 0 THEN
		Initializable[i] := Initialize;
		InitializableCount := InitializableCount + 1;
		EXIT;
	END_IF
END_FOR
END_METHOD

{attribute 'monitoring' := 'call'}
PROPERTY Initialized : BOOL
GET
VAR
	i		   : UDINT;
	Initialize : I_Initializable;
END_VAR
Initialized := TRUE;
FOR i := 0 TO MaxCount DO
	IF Initializable[i] = 0 THEN
		EXIT;
	END_IF

	IF NOT Initializable[i].Initialized THEN
		Initialized := FALSE;
	END_IF
END_FOR
END_GET
END_PROPERTY

METHOD Initializing
VAR_INST
	Logged : BOOL;
END_VAR

VAR
	i		   : UDINT;
	Initialize : I_Initializable;
END_VAR
FOR i := 0 TO MaxCount DO
	IF Initializable[i] = 0 THEN
		RETURN;
	END_IF

	Initializable[i].Initialize();
END_FOR

IF NOT Logged THEN
	Logged := TRUE;
	Trace.LogMessage('Initializer', 'Collection is full. Review library parameters and code to ensure proper setup.');
END_IF
END_METHOD

METHOD RemoveInitialize : RegistrationResult
VAR_INPUT
	Initialize : I_Initializable;
END_VAR

VAR
	i : UDINT;
	PresentInCollection : BOOL;
END_VAR
IF Initialize = 0 THEN
	RemoveInitialize := RegistrationResult.NullReference;
	RETURN;
END_IF

IF InitializableCount = 0 THEN
	RemoveInitialize := RegistrationResult.CollectionEmpty;
	RETURN;
END_IF

FOR i := 0 TO MaxCount DO
	IF Initializable[i] = Initialize THEN
		PresentInCollection := TRUE;
	END_IF
END_FOR

IF NOT PresentInCollection THEN
	RemoveInitialize := RegistrationResult.NotFoundInCollection;
	RETURN;
END_IF

FOR i := 0 TO MaxCount DO
	IF Initializable[i] = Initialize THEN
		InitializableCount := InitializableCount - 1;
		IF i < MaxCount THEN
			MEMMOVE(ADR(Initializable[i]), ADR(Initializable[i + 1]), (MaxCount - i) * SIZEOF(Initialize));
		ELSE
			Initializable[MaxCount] := 0;
		END_IF

		EXIT;
	END_IF
END_FOR
END_METHOD

END_FUNCTION_BLOCK

// _Internal/List/Interface/I_List
INTERFACE I_List EXTENDS I_Collection

METHOD ContainsItem : BOOL
VAR_INPUT
	Item : I_Base;
	;
END_VAR
END_METHOD

METHOD GetAtIndex : I_Base
VAR_INPUT
	Index : UDINT;
END_VAR
END_METHOD

METHOD InsertAtIndex : BOOL
VAR_INPUT
	Item  : I_Base;
	Index : UDINT;
END_VAR
END_METHOD

METHOD RemoveAtIndex
VAR_INPUT
	Index : UDINT;
END_VAR
END_METHOD

END_INTERFACE

// _Internal/List/List
FUNCTION_BLOCK List
VAR_GENERIC CONSTANT
	ListSize : UDINT := 2;
END_VAR
EXTENDS Collection<ListSize> IMPLEMENTS I_List
VAR
	_ListCount : UDINT := 0;
END_VAR

METHOD AddItem
VAR_INPUT
	Item : I_Base;
END_VAR
SUPER^.AddItem(Item);
CountListItems();
END_METHOD

METHOD Clear
SUPER^.Clear();
CountListItems();
END_METHOD

METHOD RemoveItem
VAR_INPUT
	Item : I_Base;
END_VAR

VAR
	pItem		 : POINTER TO I_Base;
	pItemNext	 : POINTER TO I_Base;
	i			 : UDINT;
	removedItems : UDINT;
END_VAR
IF _Count = 0 THEN
	Trace.LogMessage(InstancePath, 'No Items found in this Collection!');
	RETURN;
END_IF

IF Item = 0 THEN
	Trace.LogMessage(InstancePath, 'Item to remove needs to be valid interface!');
	RETURN;
END_IF

FOR i := 0 TO (_Count - 1) DO
	IF _Data[i] = Item THEN
		_Data[i]	 := 0;
		removedItems := removedItems + 1;
	END_IF
END_FOR

IF _Count > 1 THEN
	FOR i := 0 TO (_Count - 2) DO
		IF _Data[i] = 0 AND _Data[i + 1] <> 0 THEN
			_Data[i]	 := _Data[i + 1];
			_Data[i + 1] := 0;
		END_IF
	END_FOR
END_IF

CountListItems();
_Count := _Count - removedItems;
END_METHOD

METHOD PRIVATE CountListItems
VAR
	i	  : UDINT;
	pItem : POINTER TO I_Base;
END_VAR
IF _Count = 0 THEN
	_ListCount := 0;
	RETURN;
END_IF

_ListCount := 0;
FOR i := 0 TO (_Count - 1) DO
	IF _Data[i] <> 0 THEN
		_ListCount := _ListCount + 1;
	END_IF
END_FOR
END_METHOD

METHOD ContainsItem : BOOL
VAR_INPUT
	Item : I_Base;
END_VAR

VAR
	i	  : UDINT;
	pItem : POINTER TO I_Base;
END_VAR
IF Item = 0 THEN
	Trace.LogMessage(InstancePath, 'Item is not a valid interface!');
	RETURN;
END_IF

IF _ListCount = 0 THEN
	RETURN;
END_IF

FOR i := 0 TO (_ListCount - 1) DO
	IF _Data[i] = Item AND _Data[i] <> 0 THEN
		ContainsItem := TRUE;
		RETURN;
	END_IF
END_FOR
END_METHOD

{attribute 'monitoring' := 'call'}
PROPERTY Count : UDINT
GET
Count := _ListCount;
END_GET
END_PROPERTY

METHOD GetAtIndex : I_Base
VAR_INPUT
	Index : UDINT;
END_VAR

VAR
	pItem : POINTER TO I_Base;
END_VAR
IF Count = 0 THEN
	Trace.LogMessage(InstancePath, 'No Items found in this List!');
	RETURN;
END_IF

IF Index > (_Count - 1) THEN
	Trace.LogMessage(InstancePath, 'Index does not exist in List!');
	RETURN;
END_IF

GetAtIndex := _Data[Index];
END_METHOD

METHOD InsertAtIndex : BOOL
VAR_INPUT
	Item  : I_Base;
	Index : UDINT;
END_VAR

VAR
	pItem	  : POINTER TO I_Base;
	pItemNext : POINTER TO I_Base;
	i		  : UDINT;
END_VAR
IF Index > _Count THEN
	InsertAtIndex := FALSE;
	RETURN;
END_IF

_Count := (_Count + 1);
FOR i := _Count TO Index + 1 BY -1 DO
	_Data[i] := _Data[i - 1];
END_FOR

_Data[Index] := Item;
CountListItems();
END_METHOD

METHOD RemoveAtIndex
VAR_INPUT
	Index : UDINT;
END_VAR

VAR
	pItem : POINTER TO I_Base;
END_VAR
IF Count = 0 THEN
	Trace.LogMessage(InstancePath, 'No Items found in this List!');
	RETURN;
END_IF

IF Index > (_Count - 1) THEN
	Trace.LogMessage(InstancePath, 'Index does not exist in List!');
	RETURN;
END_IF

MEMMOVE(ADR(_Data[Index]), ADR(_Data[Index + 1]), (_Count - Index - 1) * SIZEOF(PVOID));
_Count := _Count - 1;

//pItem  := Collection.pBuffer + (Index * SIZEOF(PVOID));
CountListItems();
END_METHOD

END_FUNCTION_BLOCK

// _Internal/Module/Interface/I_ContainModules
INTERFACE I_ContainModules

METHOD DeregisterCyclic : RegistrationResult
VAR_INPUT
	Cyclic : I_Cyclic;
END_VAR
END_METHOD

METHOD DeregisterInitialize : RegistrationResult
VAR_INPUT
	Initializable : I_Initializable;
END_VAR
END_METHOD

METHOD DeregisterModule : RegistrationResult
VAR_INPUT
	Module : I_Module;
END_VAR
END_METHOD

PROPERTY Modules : I_ModuleCollection
GET
END_GET
END_PROPERTY

METHOD RegisterCyclic  : RegistrationResult
VAR_INPUT
	Cyclic : I_Cyclic;
END_VAR
END_METHOD

METHOD RegisterInitialize  : RegistrationResult
VAR_INPUT
	Initializable : I_Initializable;
END_VAR
END_METHOD

METHOD RegisterModule  : RegistrationResult
VAR_INPUT
	Module : I_Module;
END_VAR
END_METHOD

END_INTERFACE

// Module/Module
FUNCTION_BLOCK ABSTRACT Module IMPLEMENTS I_Module, I_Cyclic, I_Initializable
VAR
	_Name				: T_MaxString;
	ModuleInitialized	: BOOL;
	CyclicRunner		: CyclicRunner<CoreParameter.MaxCountInCollections>;
	ComponentCollection : ComponentCollection<CoreParameter.MaxCountInCollections>;
	ModuleCollection	: ModuleCollection<CoreParameter.MaxCountInCollections>;
	Initializer			: Initializer<CoreParameter.MaxCountInCollections>;
END_VAR

//FB_Init is always available implicitly and it is used primarily for initialization.

//The return value is not evaluated. For a specific influence, you can also declare the

//methods explicitly and provide additional code there with the standard initialization

//code. You can evaluate the return value.
METHOD FB_Init : BOOL
VAR_INPUT
	bInitRetains : BOOL; // TRUE: the retain variables are initialized (reset warm / reset cold)
	bInCopyCode	 : BOOL; // TRUE: the instance will be copied to the copy code afterward (online change)   
	Name		 : T_MaxString;
END_VAR
_Name := Name;
END_METHOD

METHOD CyclicLogic
OnCyclicCall();
CyclicRunner.CallAll();
END_METHOD

METHOD ABSTRACT OnCyclicCall
VAR_INPUT
END_VAR
END_METHOD

METHOD DeregisterComponent : RegistrationResult
VAR_INPUT
	Component : I_Component;
END_VAR
DeregisterComponent := ComponentCollection.RemoveComponent(Component);
END_METHOD

METHOD DeregisterCyclic : RegistrationResult
VAR_INPUT
	Cyclic : I_Cyclic;
END_VAR
DeregisterCyclic := CyclicRunner.RemoveCallee(Cyclic);
END_METHOD

METHOD DeregisterInitialize : RegistrationResult
VAR_INPUT
	Initializable : I_Initializable;
END_VAR
DeregisterInitialize := Initializer.RemoveInitialize(Initializable);
END_METHOD

METHOD DeregisterModule : RegistrationResult
VAR_INPUT
	Module : I_Module;
END_VAR
DeregisterModule := ModuleCollection.RemoveModule(Module);
END_METHOD

METHOD DeregisterWithParent
VAR_INPUT
	Parent : I_ContainModules;
END_VAR
Parent.DeregisterModule(THIS^);
Parent.DeregisterCyclic(THIS^);
Parent.DeregisterInitialize(THIS^);
END_METHOD

METHOD Initialize
IF NOT ModuleInitialized THEN
	Initializing();
	RETURN;
END_IF

Initializer.Initializing();
END_METHOD

{attribute 'monitoring' := 'call'}
PROPERTY Initialized : BOOL
GET
Initialized := ModuleInitialized AND Initializer.Initialized;
END_GET
SET
ModuleInitialized := Initialized;
END_SET
END_PROPERTY

(* This Module will be done initialize when ModuleInitialized := TRUE;, subequently all subitems will be called to be initialized *)
METHOD ABSTRACT Initializing
// ModuleInitialized := TRUE;
END_METHOD

METHOD RegisterComponent : RegistrationResult
VAR_INPUT
	Component : I_Component;
END_VAR
RegisterComponent := ComponentCollection.AddComponent(Component);
END_METHOD

METHOD RegisterCyclic : RegistrationResult
VAR_INPUT
	Cyclic : I_Cyclic;
END_VAR
RegisterCyclic := CyclicRunner.AddCallee(Cyclic);
END_METHOD

METHOD RegisterInitialize : RegistrationResult
VAR_INPUT
	Initializable : I_Initializable;
END_VAR
RegisterInitialize := Initializer.AddInitialize(Initializable);
END_METHOD

METHOD RegisterModule : RegistrationResult
VAR_INPUT
	Module : I_Module;
END_VAR
RegisterModule := ModuleCollection.AddModule(Module);
END_METHOD

METHOD RegisterWithParent
VAR_INPUT
	Parent : I_ContainModules;
END_VAR
Parent.RegisterModule(THIS^);
Parent.RegisterCyclic(THIS^);
Parent.RegisterInitialize(THIS^);
END_METHOD

METHOD ResetComponents : BOOL
VAR_INST
	ResetComponentsVisitor : ResetComponentsVisitor;
END_VAR
ResetComponentsVisitor.Reset(THIS^);
ResetComponents := NOT ResetComponentsVisitor.Error AND NOT ResetComponentsVisitor.Busy;
END_METHOD

METHOD ResetModules : BOOL
VAR_INST
	ResetModulesVisitor : ResetModulesVisitor;
END_VAR
ResetModulesVisitor.Reset(THIS^);
ResetModules := NOT ResetModulesVisitor.Error AND NOT ResetModulesVisitor.Busy;
END_METHOD

METHOD Accept
VAR_INPUT
	Visitor : I_ModuleVisitor;
END_VAR
Visitor.VisitModule(THIS^);
END_METHOD

PROPERTY Components : I_ComponentCollection
GET
Components := ComponentCollection;
END_GET
END_PROPERTY

PROPERTY Modules : I_ModuleCollection
GET
Modules := ModuleCollection;
END_GET
END_PROPERTY

{attribute 'monitoring' := 'call'}
PROPERTY Name : T_MaxString
GET
Name := _Name;
END_GET
SET
_Name := Name;
END_SET
END_PROPERTY

END_FUNCTION_BLOCK

// Module/Interface/I_Module
INTERFACE I_Module EXTENDS I_ContainComponents, I_ContainModules, I_Base

METHOD Accept
VAR_INPUT
	Visitor : I_ModuleVisitor;
END_VAR
END_METHOD

METHOD DeregisterWithParent
VAR_INPUT
	Parent : I_ContainModules;
END_VAR
END_METHOD

{attribute 'monitoring' := 'call'}
PROPERTY Name : T_MaxString
GET
END_GET
END_PROPERTY

METHOD RegisterWithParent
VAR_INPUT
	Parent : I_ContainModules;
END_VAR
END_METHOD

METHOD ResetComponents : BOOL
END_METHOD

METHOD ResetModules : BOOL
END_METHOD

END_INTERFACE

// Module/Interface/I_ModuleVisitor
INTERFACE I_ModuleVisitor

METHOD VisitModule
VAR_INPUT
	Module : I_Module;
END_VAR
END_METHOD

END_INTERFACE

// _Internal/Module/ModuleCollection
FUNCTION_BLOCK ModuleCollection
VAR_GENERIC CONSTANT
	MaxCount : UDINT := 10;
END_VAR IMPLEMENTS I_ModuleCollection
VAR
	Modules		: ARRAY[0..MaxCount] OF I_Module;
	ModuleCount : UDINT;
	NullModule	: NullModule('Null Module');
END_VAR

METHOD Accept
VAR_INPUT
	Visitor : I_ModuleVisitor;
END_VAR

VAR
	i : UDINT;
END_VAR
FOR i := 0 TO MaxCount DO
	IF Modules[i] = 0 THEN
		EXIT;
	END_IF

	Modules[i].Accept(Visitor);
END_FOR
END_METHOD

METHOD AddModule : RegistrationResult
VAR_INPUT
	Module : I_Module;
END_VAR

VAR
	i : UDINT;
	Registered : BOOL;
END_VAR
IF Module = 0 THEN
	AddModule := RegistrationResult.NullReference;
	RETURN;
END_IF

IF ModuleCount >= MaxCount THEN
	AddModule := RegistrationResult.TooManyComponents;
	RETURN;
END_IF

FOR i := 0 TO MaxCount DO
	IF Modules[i] = Module THEN
		Registered := TRUE;
	END_IF
END_FOR

IF Registered THEN
	AddModule := RegistrationResult.AlreadyAdded;
	RETURN;
END_IF

FOR i := 0 TO MaxCount DO
	IF Modules[i] = 0 THEN
		Modules[i] := Module;
		ModuleCount := ModuleCount + 1;
		EXIT;
	END_IF
END_FOR
END_METHOD

{attribute 'monitoring' := 'call'}
PROPERTY Count : UDINT
GET
Count := TO_UDINT(ModuleCount);
END_GET
END_PROPERTY

METHOD GetAtIndex : I_Module
VAR_INPUT
	Index : UDINT;
END_VAR
IF Index > Count THEN
	GetAtIndex := NullModule;
	RETURN;
END_IF

IF Index < 0 THEN
	GetAtIndex := NullModule;
	RETURN;
END_IF

IF Modules[Index] <> 0 THEN
	GetAtIndex := Modules[Index];
ELSE
	GetAtIndex := NullModule;
END_IF
END_METHOD

METHOD GetModuleByName : I_Module
VAR_INPUT
	Name : T_MaxString;
END_VAR

VAR
	i : UDINT;
END_VAR
FOR i := 0 TO MaxCount DO
	IF Modules[i] = 0 THEN
		EXIT;
	END_IF

	IF Modules[i].Name = Name THEN
		GetModuleByName := Modules[i];
		EXIT;
	END_IF
END_FOR
END_METHOD

METHOD RemoveModule : RegistrationResult
VAR_INPUT
	Module : I_Module;
END_VAR

VAR
	i : UDINT;
	PresentInCollection : BOOL;
END_VAR
IF Module = 0 THEN
	RemoveModule := RegistrationResult.NullReference;
	RETURN;
END_IF

IF ModuleCount = 0 THEN
	RemoveModule := RegistrationResult.CollectionEmpty;
	RETURN;
END_IF

FOR i := 0 TO MaxCount DO
	IF Modules[i] = Module THEN
		PresentInCollection := TRUE;
	END_IF
END_FOR

IF NOT PresentInCollection THEN
	RemoveModule := RegistrationResult.NotFoundInCollection;
	RETURN;
END_IF

FOR i := 0 TO MaxCount DO
	IF Modules[i] = Module THEN
		IF i < MaxCount THEN
			MEMMOVE(ADR(Modules[i]), ADR(Modules[i + 1]), (MaxCount - i) * SIZEOF(Module));
		ELSE
			Modules[MaxCount] := 0;
		END_IF

		EXIT;
	END_IF
END_FOR
END_METHOD

END_FUNCTION_BLOCK

// _Internal/Module/Interface/I_ModuleCollection
INTERFACE I_ModuleCollection

METHOD Accept
VAR_INPUT
	Visitor : I_ModuleVisitor;
END_VAR
END_METHOD

{attribute 'monitoring' := 'call'}
PROPERTY Count : UDINT
GET
END_GET
END_PROPERTY

METHOD GetAtIndex : I_Module
VAR_INPUT
	Index : UDINT;
END_VAR
END_METHOD

METHOD GetModuleByName : I_Module
VAR_INPUT
	Name : T_MaxString;
END_VAR
END_METHOD

END_INTERFACE

// _Internal/Null/NullModule
FUNCTION_BLOCK NullModule IMPLEMENTS I_Module
VAR
    _Name : T_MaxString;
END_VAR

METHOD Accept
VAR_INPUT
	Visitor	: I_ModuleVisitor;
END_VAR
END_METHOD

PROPERTY Components : I_ComponentCollection
GET
END_GET
END_PROPERTY

METHOD DeregisterComponent : RegistrationResult
VAR_INPUT
	Component	: I_Component;
END_VAR
END_METHOD

METHOD DeregisterCyclic : RegistrationResult
VAR_INPUT
	Cyclic	: I_Cyclic;
END_VAR
END_METHOD

METHOD DeregisterInitialize : RegistrationResult
VAR_INPUT
	Initializable	: I_Initializable;
END_VAR
END_METHOD

METHOD DeregisterModule : RegistrationResult
VAR_INPUT
	Module	: I_Module;
END_VAR
END_METHOD

METHOD DeregisterWithParent
VAR_INPUT
	Parent	: I_ContainModules;
END_VAR
END_METHOD

//FB_Init is always available implicitly and it is used primarily for initialization.

//The return value is not evaluated. For a specific influence, you can also declare the

//methods explicitly and provide additional code there with the standard initialization

//code. You can evaluate the return value.
METHOD FB_Init : BOOL
VAR_INPUT
	bInitRetains : BOOL; // TRUE: the retain variables are initialized (reset warm / reset cold)
	bInCopyCode	 : BOOL; // TRUE: the instance will be copied to the copy code afterward (online change)   
	Name		 : T_MaxString;
END_VAR
_Name := Name;
END_METHOD

PROPERTY Modules : I_ModuleCollection
GET
END_GET
END_PROPERTY

{attribute 'monitoring' := 'call'}
PROPERTY Name : T_MaxString
GET
Name := _Name;
END_GET
SET
_Name := Name;
END_SET
END_PROPERTY

METHOD RegisterComponent : RegistrationResult
VAR_INPUT
	Component	: I_Component;
END_VAR
END_METHOD

METHOD RegisterCyclic : RegistrationResult
VAR_INPUT
	Cyclic	: I_Cyclic;
END_VAR
END_METHOD

METHOD RegisterInitialize : RegistrationResult
VAR_INPUT
	Initializable	: I_Initializable;
END_VAR
END_METHOD

METHOD RegisterModule : RegistrationResult
VAR_INPUT
	Module	: I_Module;
END_VAR
END_METHOD

METHOD RegisterWithParent
VAR_INPUT
	Parent	: I_ContainModules;
END_VAR
END_METHOD

METHOD ResetComponents : BOOL
END_METHOD

METHOD ResetModules : BOOL
END_METHOD

END_FUNCTION_BLOCK

// Visitors/Reset/ResetComponentsVisitor
FUNCTION_BLOCK ResetComponentsVisitor IMPLEMENTS I_ComponentVisitor, I_TaskResult
VAR
	{attribute 'hide'}
	Resettable : I_Resettable;
	{attribute 'hide'}
	Result : I_TaskResult;
	{attribute 'hide'}
	_Busy : BOOL;
	{attribute 'hide'}
	_Error : BOOL;
	{attribute 'hide'}
	_ErrorId	   : UDINT;
	ErrorComponent : I_Component;
END_VAR

{attribute 'monitoring' := 'call'}
PROPERTY Busy : BOOL
GET
Busy := _Busy;
END_GET
END_PROPERTY

{attribute 'monitoring' := 'call'}
PROPERTY Error : BOOL
GET
Error := _Error;
END_GET
END_PROPERTY

{attribute 'monitoring' := 'call'}
PROPERTY ErrorId : UDINT
GET
ErrorID := _ErrorID;
END_GET
END_PROPERTY

METHOD Reset
VAR_INPUT
	Module : I_Module;
END_VAR
_Error	 := FALSE;
_ErrorId := 0;
_Busy	 := FALSE;
Module.Components.Accept(THIS^);
END_METHOD

METHOD VisitComponent
VAR_INPUT
	Component : I_Component;
END_VAR
IF __QUERYINTERFACE(Component, Resettable) THEN
	Resettable.Reset();
END_IF

IF __QUERYINTERFACE(Component, Result) THEN
	IF Result.Error THEN
		ErrorComponent := Component;
		_Error		   := TRUE;
		_ErrorId	   := Result.ErrorId;
	END_IF

	IF Result.Busy THEN
		_Busy := TRUE;
	END_IF
END_IF
END_METHOD

END_FUNCTION_BLOCK

// Visitors/Reset/ResetModulesVisitor
FUNCTION_BLOCK ResetModulesVisitor IMPLEMENTS I_ModuleVisitor, I_TaskResult
VAR
	{attribute 'hide'}
	Resettable : I_Resettable;
	{attribute 'hide'}
	Result : I_TaskResult;
	{attribute 'hide'}
	_Busy : BOOL;
	{attribute 'hide'}
	_Error : BOOL;
	{attribute 'hide'}
	_ErrorId	: UDINT;
	ErrorModule : I_Module;
END_VAR

{attribute 'monitoring' := 'call'}
PROPERTY Busy : BOOL
GET
Busy := _Busy;
END_GET
END_PROPERTY

{attribute 'monitoring' := 'call'}
PROPERTY Error : BOOL
GET
Error := _Error;
END_GET
END_PROPERTY

{attribute 'monitoring' := 'call'}
PROPERTY ErrorId : UDINT
GET
ErrorID := _ErrorID;
END_GET
END_PROPERTY

METHOD Reset
VAR_INPUT
	Module : I_Module;
END_VAR
_Error	 := FALSE;
_ErrorId := 0;
_Busy	 := FALSE;
Module.Modules.Accept(THIS^);
END_METHOD

METHOD VisitModule
VAR_INPUT
	Module : I_Module;
END_VAR
IF __QUERYINTERFACE(Module, Resettable) THEN
	Resettable.Reset();
END_IF

IF __QUERYINTERFACE(Module, Result) THEN
	IF Result.Error THEN
		ErrorModule := Module;
		_Error		:= TRUE;
		_ErrorId	:= Result.ErrorId;
	END_IF

	IF Result.Busy THEN
		_Busy := TRUE;
	END_IF
END_IF
END_METHOD

END_FUNCTION_BLOCK

// _Internal/Statemachine/Interface/I_StateList
INTERFACE I_StateList

METHOD AddStateAtIndex
VAR_INPUT
	Index : DINT;
	State : I_State;
END_VAR
END_METHOD

METHOD GetStateAtIndex : I_State
VAR_INPUT
	Index : DINT;
END_VAR
END_METHOD

PROPERTY NumberOfStates : DINT
GET
END_GET
END_PROPERTY

END_INTERFACE

// Statemachine/Generic/State
FUNCTION_BLOCK ABSTRACT State IMPLEMENTS I_State
VAR
	Statemachine  : I_Statemachine;
	SequenceState : UDINT;
END_VAR

METHOD Executing : BOOL
Executing := TRUE;
END_METHOD

//FB_Init is always available implicitly and it is used primarily for initialization.

//The return value is not evaluated. For a specific influence, you can also declare the

//methods explicitly and provide additional code there with the standard initialization

//code. You can evaluate the return value.
METHOD FB_Init : BOOL
VAR_INPUT
	bInitRetains : BOOL; // TRUE: the retain variables are initialized (reset warm / reset cold)
	bInCopyCode	 : BOOL; // TRUE: the instance will be copied to the copy code afterward (online change)  
	State		 : DINT;
	Statemachine : I_Statemachine;
END_VAR
THIS^.Statemachine := Statemachine;
IF THIS^.Statemachine <> 0 THEN
	THIS^.Statemachine.States.AddStateAtIndex(State, THIS^);
END_IF
END_METHOD

METHOD Inactive
SequenceState := 0;
END_METHOD

END_FUNCTION_BLOCK

// Statemachine/Interface/I_State
INTERFACE I_State EXTENDS I_Base

METHOD Executing : BOOL;
END_METHOD

METHOD Inactive
VAR_INPUT
END_VAR
END_METHOD

END_INTERFACE

// Statemachine/Generic/Statemachine
FUNCTION_BLOCK Statemachine
VAR_GENERIC CONSTANT
	InitialState : DINT := 1;
END_VAR
EXTENDS CyclicComponent IMPLEMENTS I_Statemachine
VAR
	StateList	  : StateList<TO_DINT(CoreParameter.MaxCountInCollections)>;
	_CurrentState : DINT := InitialState;
	{attribute 'hide'}
	DefaultModeController : ModeControl;
	_Mode				  : I_Mode := DefaultModeController;
END_VAR

PROPERTY Mode : I_Mode
GET
Mode := _Mode;
END_GET
SET
_Mode := Mode;
END_SET
END_PROPERTY

METHOD ChangeState
VAR_INPUT
	StateCommand : DINT;
END_VAR
IF StateList.NumberOfStates = 0 THEN
	Trace.LogMessage('Statemachine', 'No states defined!');
	RETURN;
END_IF

_CurrentState := StateCommand;
END_METHOD

{attribute 'monitoring' := 'call'}
PROPERTY CurrentState : DINT
GET
CurrentState := _CurrentState;
END_GET
END_PROPERTY

PROPERTY States : I_StateList
GET
States := StateList;
END_GET
END_PROPERTY

METHOD CyclicLogic
VAR
	i	  : DINT;
	State : I_State;
END_VAR
IF StateList.NumberOfStates = 0 THEN
	RETURN;
END_IF

FOR i := 0 TO (StateList.NumberOfStates - 1) DO
	State := StateList.GetStateAtIndex(i);
	IF State <> 0 THEN
		IF (i = _CurrentState) THEN
			State.Executing();
		ELSE
			State.Inactive();
		END_IF
	END_IF
END_FOR
END_METHOD

END_FUNCTION_BLOCK

// Component/CyclicComponent
FUNCTION_BLOCK ABSTRACT CyclicComponent EXTENDS Component IMPLEMENTS I_Cyclic
VAR
	RegisteredAsCyclicResult : RegistrationResult;
END_VAR

METHOD ABSTRACT CyclicLogic
END_METHOD

METHOD DeregisterWithParent
VAR_INPUT
	Parent : I_ContainComponents;
END_VAR
Parent.DeregisterComponent(THIS^);
Parent.DeregisterCyclic(THIS^);
END_METHOD

METHOD RegisterWithParent
VAR_INPUT
	Parent : I_ContainComponents;
END_VAR
RegisteredAsComponentResult := Parent.RegisterComponent(THIS^);
RegisteredAsCyclicResult := Parent.RegisterCyclic(THIS^);
END_METHOD

END_FUNCTION_BLOCK

// Statemachine/Interface/I_Statemachine
INTERFACE I_Statemachine EXTENDS I_Component

METHOD ChangeState
VAR_INPUT
	StateCommand : DINT;
END_VAR
END_METHOD

{attribute 'monitoring' := 'call'}
PROPERTY CurrentState : DINT
GET
END_GET
END_PROPERTY

PROPERTY Mode : I_Mode
GET
END_GET
SET
END_SET
END_PROPERTY

PROPERTY States : I_StateList
GET
END_GET
END_PROPERTY

END_INTERFACE

// Modes/Interface/I_Mode
INTERFACE I_Mode EXTENDS I_Base

METHOD ChangeMode
VAR_INPUT
	RequestedMode : DINT;
END_VAR
END_METHOD

{attribute 'monitoring' := 'call'}
PROPERTY CurrentMode : DINT
GET
END_GET
END_PROPERTY

END_INTERFACE

// _Internal/Statemachine/StateList
FUNCTION_BLOCK StateList
VAR_GENERIC CONSTANT
	MaxCount : DINT := 10;
END_VAR IMPLEMENTS I_StateList
VAR
	States : ARRAY[0..MaxCount] OF I_State;
END_VAR

METHOD AddStateAtIndex
VAR_INPUT
	Index : DINT;
	State : I_State;
END_VAR
IF Index > MaxCount THEN
	RETURN;
END_IF

States[Index] := State;
END_METHOD

METHOD GetStateAtIndex : I_State
VAR_INPUT
	Index : DINT;
END_VAR
IF Index > MaxCount THEN
	RETURN;
END_IF

GetStateAtIndex := States[Index];
END_METHOD

PROPERTY NumberOfStates : DINT
GET
NumberOfStates := MaxCount;
END_GET
END_PROPERTY

END_FUNCTION_BLOCK

// Modes/ModeControl
FUNCTION_BLOCK ModeControl IMPLEMENTS I_Mode
VAR
	{attribute 'hide'}
	_CurrentMode : DINT := 1;
END_VAR

METHOD ChangeMode
VAR_INPUT
	RequestedMode : DINT;
END_VAR
IF (RequestedMode >= 1) THEN
	_CurrentMode := RequestedMode;
ELSE
	Trace.LogMessage('Mode Controller', 'Requested Mode is not Defined');
END_IF
END_METHOD

{attribute 'monitoring' := 'call'}
PROPERTY CurrentMode : DINT
GET
CurrentMode := _CurrentMode;
END_GET
END_PROPERTY

END_FUNCTION_BLOCK

// _Internal/Tracing/Interface/I_ContainTraceArgument
INTERFACE I_ContainTraceArgument EXTENDS I_Base

{attribute 'monitoring' := 'call'}
PROPERTY Arguments : I_TraceArgument
GET
END_GET
END_PROPERTY

END_INTERFACE

// _Internal/Tracing/Interface/I_TraceArgument
INTERFACE I_TraceArgument EXTENDS I_Base, I_ToString

END_INTERFACE

// _Internal/Tracing/Interface/I_ContainTracePublisher
INTERFACE I_ContainTracePublisher EXTENDS I_Base

PROPERTY Publisher : I_TracePublisher
GET
END_GET
END_PROPERTY

END_INTERFACE

// _Internal/Tracing/Interface/I_TraceInstanceLogger
INTERFACE I_TraceInstanceLogger EXTENDS I_Base

METHOD LogMessageInstance
VAR_INPUT
	SourceInfo	: I_TraceSourceInfo;
	MessageInfo : I_TraceMessageInfo;
	Arguments	: I_TraceArgument := 0;
END_VAR
END_METHOD

END_INTERFACE

// _Internal/Tracing/Interface/I_TraceSourceInfo
INTERFACE I_TraceSourceInfo EXTENDS I_Base

{attribute 'monitoring':='call'}
PROPERTY SourceId : UDINT
GET
END_GET
END_PROPERTY

{attribute 'monitoring':='call'}
PROPERTY SourceName : T_MaxString
GET
END_GET
END_PROPERTY

{attribute 'monitoring':='call'}
PROPERTY TimeStamp : ULINT
GET
END_GET
END_PROPERTY

END_INTERFACE

// _Internal/Tracing/Interface/I_TraceMessageInfo
INTERFACE I_TraceMessageInfo EXTENDS I_Base

{attribute 'monitoring':='call'}
PROPERTY Message : T_MaxString
GET
END_GET
END_PROPERTY

{attribute 'monitoring':='call'}
PROPERTY MessageId : UDINT
GET
END_GET
END_PROPERTY

{attribute 'monitoring':='call'}
PROPERTY Severity : USINT
GET
END_GET
END_PROPERTY

END_INTERFACE

// _Internal/Tracing/AdsLogger
FUNCTION_BLOCK AdsLogger IMPLEMENTS I_TraceLogger
VAR
	MessagesThisScan : DINT;
	CurrentCycle	 : UDINT;
END_VAR

//FB_Init is always available implicitly and it is used primarily for initialization.

//The return value is not evaluated. For a specific influence, you can also declare the

//methods explicitly and provide additional code there with the standard initialization

//code. You can evaluate the return value.
METHOD FB_Init : BOOL
VAR_INPUT
	bInitRetains   : BOOL; // TRUE: the retain variables are initialized (reset warm / reset cold)
	bInCopyCode	   : BOOL; // TRUE: the instance will be copied to the copy code afterward (online change)   
	TracePublisher : I_TracePublisher;
END_VAR
IF CoreParameter.EnableAdsLogger THEN
	TracePublisher.Subscribe(THIS^);
END_IF
END_METHOD

METHOD LogMessage
VAR_INPUT
	Key		  : T_MaxString;
	Value	  : T_MaxString;
	SourceId  : UDINT := 0;
	TimeStamp : ULINT := 0;
	MessageId : UDINT := 1;
	Severity  : USINT := 1;
END_VAR
IF GETCURTASKINDEXEX() > 0 THEN
	IF TwinCAT_SystemInfoVarList._TaskInfo[GETCURTASKINDEXEX()].CycleCount <> CurrentCycle THEN
		CurrentCycle	 := TwinCAT_SystemInfoVarList._TaskInfo[GETCURTASKINDEXEX()].CycleCount;
		MessagesThisScan := 0;
	END_IF

	IF NOT (MessagesThisScan < TO_DINT(TwinCAT_SystemInfoVarList._TaskInfo[GETCURTASKINDEXEX()].CycleTime / 2000)) THEN
		RETURN;
	END_IF
END_IF

CASE Severity OF
	0, 1:
		ADSLOGSTR(ADSLOG_MSGTYPE_LOG OR ADSLOG_MSGTYPE_HINT, Concat(Value, ': %s'), Key);

	2:
		ADSLOGSTR(ADSLOG_MSGTYPE_LOG OR ADSLOG_MSGTYPE_WARN, Concat(Value, ': %s'), Key);

	3, 4:
		ADSLOGSTR(ADSLOG_MSGTYPE_LOG OR ADSLOG_MSGTYPE_ERROR, Concat(Value, ': %s'), Key);
END_CASE

MessagesThisScan := MessagesThisScan + 1;
END_METHOD

END_FUNCTION_BLOCK

// _Internal/Tracing/TcEventLogger
FUNCTION_BLOCK TcEventLogger IMPLEMENTS I_TraceLogger
VAR
	MessagesThisScan : DINT;
	Message			 : FB_TcMessage;
	Source			 : FB_TcSourceInfo;
	CurrentCycle	 : UDINT;
END_VAR

//FB_Init is always available implicitly and it is used primarily for initialization.

//The return value is not evaluated. For a specific influence, you can also declare the

//methods explicitly and provide additional code there with the standard initialization

//code. You can evaluate the return value.
METHOD FB_Init : BOOL
VAR_INPUT
	bInitRetains   : BOOL; // TRUE: the retain variables are initialized (reset warm / reset cold)
	bInCopyCode	   : BOOL; // TRUE: the instance will be copied to the copy code afterward (online change)   
	TracePublisher : I_TracePublisher;
END_VAR
IF CoreParameter.EnableTcEventLogging THEN
	TracePublisher.Subscribe(THIS^);
END_IF
END_METHOD

METHOD LogMessage
VAR_INPUT
	Key		  : T_MaxString;
	Value	  : T_MaxString;
	SourceId  : UDINT := 0;
	TimeStamp : ULINT := 0;
	MessageId : UDINT := 1;
	Severity  : USINT := 1;
END_VAR
IF GETCURTASKINDEXEX() > 0 THEN
	IF TwinCAT_SystemInfoVarList._TaskInfo[GETCURTASKINDEXEX()].CycleCount <> CurrentCycle THEN
		CurrentCycle	 := TwinCAT_SystemInfoVarList._TaskInfo[GETCURTASKINDEXEX()].CycleCount;
		MessagesThisScan := 0;
	END_IF

	IF NOT (MessagesThisScan < TO_DINT(TwinCAT_SystemInfoVarList._TaskInfo[GETCURTASKINDEXEX()].CycleTime / 2000)) THEN
		RETURN;
	END_IF
END_IF

Source.sName := Key;
Source.nId	 := SourceId;
Message.Create(eventClass	:= TC_EVENT_CLASSES.Trace,
			   nEventId		:= MessageId,
			   eSeverity	:= USINT_To_TcEventSeverity(Severity),
			   ipSourceInfo := Source);

Message.ipArguments.Clear().AddString(Value);
Message.Send(TimeStamp);
Message.Release();
Source.Clear();
MessagesThisScan := MessagesThisScan + 1;
END_METHOD

END_FUNCTION_BLOCK

// _Internal/Tracing/USINT_To_TcEventSeverity
FUNCTION USINT_To_TcEventSeverity : TcEventSeverity
VAR_INPUT
	Severity : USINT;
END_VAR

USINT_To_TcEventSeverity := TcEventSeverity.Verbose;
CASE Severity OF
	0: 
		USINT_To_TcEventSeverity := TcEventSeverity.Verbose;

	1:
		USINT_To_TcEventSeverity := TcEventSeverity.Info;

	2:
		USINT_To_TcEventSeverity := TcEventSeverity.Warning;

	3:
		USINT_To_TcEventSeverity := TcEventSeverity.Error;

	4:
		USINT_To_TcEventSeverity := TcEventSeverity.Critical;
END_CASE

END_FUNCTION

// _Internal/Tracing/TraceMessageInfo
{attribute 'hide_all_locals'}
FUNCTION_BLOCK TraceMessageInfo IMPLEMENTS I_TraceMessageInfo
VAR
	_Message   : T_MaxString;
	_MessageId : UDINT;
	_Severity  : USINT;
END_VAR

{attribute 'monitoring':='call'}
PROPERTY Message : T_MaxString
GET
Message := _Message;
END_GET
SET
_Message := Message;
END_SET
END_PROPERTY

{attribute 'monitoring':='call'}
PROPERTY MessageId : UDINT
GET
MessageId := _MessageId;
END_GET
SET
_MessageId := MessageId;
END_SET
END_PROPERTY

{attribute 'monitoring':='call'}
PROPERTY Severity : USINT
GET
Severity := _Severity;
END_GET
SET
_Severity := Severity;
END_SET
END_PROPERTY

END_FUNCTION_BLOCK

// _Internal/Tracing/TraceSourceInfo
{attribute 'hide_all_locals'}
FUNCTION_BLOCK TraceSourceInfo IMPLEMENTS I_TraceSourceInfo
VAR
	_SourceId	: UDINT;
	_SourceName : T_MaxString;
	_TimeStamp	: ULINT;
END_VAR

{attribute 'monitoring' := 'call'}
PROPERTY SourceId : UDINT
GET
SourceId := _SourceId;
END_GET
SET
_SourceId := SourceId;
END_SET
END_PROPERTY

{attribute 'monitoring' := 'call'}
PROPERTY SourceName : T_MaxString
GET
SourceName := _SourceName;
END_GET
SET
_SourceName := SourceName;
END_SET
END_PROPERTY

{attribute 'monitoring' := 'call'}
PROPERTY TimeStamp : ULINT
GET
TimeStamp := _TimeStamp;
END_GET
SET
_TimeStamp := TimeStamp;
END_SET
END_PROPERTY

END_FUNCTION_BLOCK

// Events/Interface/I_EventClass
INTERFACE I_EventClass EXTENDS I_EventReaction, I_Resettable

METHOD PUBLIC Arguments : I_EventArguments
VAR_INPUT
	EventId : UDINT;
END_VAR
END_METHOD

METHOD PUBLIC ClearEventById
VAR_INPUT
	EventId : UDINT;
END_VAR
END_METHOD

{attribute 'monitoring' := 'call'}
PROPERTY IsResettable : BOOL
GET
END_GET
END_PROPERTY

METHOD PUBLIC RaiseEvent
VAR_INPUT
	EventId	  : UDINT;
END_VAR
END_METHOD

METHOD ResetBySeverity : BOOL
VAR_INPUT
	Severity : UDINT;
END_VAR
END_METHOD

METHOD SetEvent
VAR_INPUT
	EventId	  : UDINT;
	Trigger	  : POINTER TO BOOL;
	AutoReset : BOOL;
END_VAR
END_METHOD

END_INTERFACE

// Events/Interface/I_EventReaction
INTERFACE I_EventReaction EXTENDS I_Resettable

METHOD GetHighestActiveEventReaction : DINT;
END_METHOD

METHOD SetEventReactions
VAR_INPUT
	Verbose	 : DINT := 0;
	Info	 : DINT := 1;
	Warning	 : DINT := 2;
	Error	 : DINT := 3;
	Critical : DINT := 4;
END_VAR
END_METHOD

END_INTERFACE

// Events/Interface/I_EventClassTcEvents
INTERFACE I_EventClassTcEvents EXTENDS I_EventClass

METHOD PUBLIC GenerateTcEvents
VAR_INPUT
	Name   : T_MaxString;
	pClass : PVOID; // ADR(TC_Events.XY) - TC Event Class in TypeSystem
	nSize  : UDINT; // SIZEOF(ST_XY) - TC Event Class in TypeSystem
END_VAR
END_METHOD

METHOD GetHighestActiveEventSeverity : TcEventSeverity
END_METHOD

END_INTERFACE

// Events/Interface/I_EventReactionTcEvents
INTERFACE I_EventReactionTcEvents EXTENDS I_EventReaction

METHOD GetHighestActiveEventSeverity : TcEventSeverity
END_METHOD

END_INTERFACE

// Events/TcEventClass
{attribute 'enable_dynamic_creation'}
FUNCTION_BLOCK TcEventClass EXTENDS CyclicComponent IMPLEMENTS I_EventClassTcEvents
VAR
	pEventClass				   : PVOID;
	pEventBuffer			   : POINTER TO PVOID;
	pEventTriggerBuffer		   : POINTER TO PVOID;
	pEventAutoResetBuffer	   : POINTER TO PVOID;
	NullEvent				   : FB_TcAlarm;
	NullBool				   : BOOL;
	NumberOfEvents			   : UDINT;
	HighestActiveEventSeverity : TcEventSeverity;
	EventReactionVerbose	   : DINT := 0;
	EventReactionInfo		   : DINT := 1;
	EventReactionWarning	   : DINT := 2;
	EventReactionError		   : DINT := 3;
	EventReactionCritical	   : DINT := 4;
	TcEventClassArguments	   : TcEventClassArguments;
END_VAR

METHOD Dispose
VAR
	i				: UDINT;
	pEvent			: POINTER TO FB_TcAlarm;
	pDispose		: POINTER TO TcEventClass;
	pEventAutoReset : POINTER TO BOOL;
END_VAR
pDispose := THIS;
FOR i := 1 TO NumberOfEvents DO
	pEvent := GetEventInstance(i);
	__DELETE(pEvent);
	pEventAutoReset := GetEventAutoResetInstance(i);
	__DELETE(pEventAutoReset);
END_FOR

__DELETE(pEventBuffer);
__DELETE(pDispose);
__DELETE(pEventTriggerBuffer);
__DELETE(pEventAutoResetBuffer);
END_METHOD

//FB_Exit must be implemented explicitly. If there is an implementation, then the

//method is called before the controller removes the code of the function block instance

//(implicit call). The return value is not evaluated.
METHOD FB_Exit : BOOL
VAR_INPUT
	bInCopyCode : BOOL; // TRUE: the exit method is called in order to leave the instance which will be copied afterwards (online change).  
END_VAR

VAR
	i				: UDINT;
	pEvent			: POINTER TO FB_TcAlarm;
	pEventAutoReset : POINTER TO BOOL;
END_VAR
FOR i := 1 TO NumberOfEvents DO
	pEvent := GetEventInstance(i);
	__DELETE(pEvent);
	pEventAutoReset := GetEventAutoResetInstance(i);
	__DELETE(pEventAutoReset);
END_FOR

__DELETE(pEventBuffer);
__DELETE(pEventTriggerBuffer);
__DELETE(pEventAutoResetBuffer);
END_METHOD

METHOD ClearEventById
VAR_INPUT
	EventId : UDINT;
END_VAR

VAR
	pEvent : POINTER TO FB_TcAlarm;
END_VAR
IF CheckEventId(EventId) THEN
	pEvent := GetEventInstance(EventId);
	IF (pEvent <> 0) THEN
		IF pEvent^.bRaised THEN
			pEvent^.Clear();
			FindActiveSeverity();
		END_IF
	END_IF
END_IF
END_METHOD

METHOD GetHighestActiveEventReaction : DINT
CASE HighestActiveEventSeverity OF
	TcEventSeverity.Verbose:
		GetHighestActiveEventReaction := EventReactionVerbose;

	TcEventSeverity.Info:
		GetHighestActiveEventReaction := EventReactionInfo;

	TcEventSeverity.Warning:
		GetHighestActiveEventReaction := EventReactionWarning;

	TcEventSeverity.Error:
		GetHighestActiveEventReaction := EventReactionError;

	TcEventSeverity.Critical:
		GetHighestActiveEventReaction := EventReactionCritical;
END_CASE
END_METHOD

METHOD GetHighestActiveEventSeverity : TcEventSeverity
GetHighestActiveEventSeverity := HighestActiveEventSeverity;
END_METHOD

{attribute 'monitoring' := 'call'}
PROPERTY IsResettable : BOOL
GET
VAR
	i		  : UDINT;
	pEvent	  : POINTER TO FB_TcAlarm;
	pTrigger  : POINTER TO BOOL;
END_VAR
IsResettable := FALSE;
FOR i := 1 TO NumberOfEvents DO
	pTrigger := GetEventTriggerInstance(i);
	IF (pTrigger <> 0) THEN
		pEvent := GetEventInstance(i);
		IF (pEvent <> 0) AND_THEN NOT pTrigger^ AND pEvent^.bRaised THEN
			IsResettable := TRUE;
		END_IF
	END_IF
END_FOR
END_GET
END_PROPERTY

METHOD RaiseEvent
VAR_INPUT
	EventId	  : UDINT;
END_VAR

VAR
	pEvent : POINTER TO FB_TcAlarm;
END_VAR
IF CheckEventId(EventId) THEN
	pEvent := GetEventInstance(EventId);
	IF (pEvent <> 0) THEN
		IF NOT pEvent^.bRaised THEN
			pEvent^.Raise();
			IF pEvent^.eSeverity > HighestActiveEventSeverity THEN
				HighestActiveEventSeverity := pEvent^.eSeverity;
			END_IF

			pEvent^.ipArguments.Clear();
		END_IF
	END_IF
END_IF
END_METHOD

METHOD ResetBySeverity : BOOL
VAR_INPUT
	Severity : UDINT;
END_VAR

VAR
	i	   : UDINT;
	pEvent : POINTER TO FB_TcAlarm;
END_VAR
FOR i := 1 TO NumberOfEvents DO
	pEvent := GetEventInstance(i);
	IF (pEvent <> 0) AND_THEN (pEvent^.eSeverity <= TO_DINT(Severity)) THEN
		pEvent^.Clear();
	END_IF
END_FOR

FindActiveSeverity();
ResetBySeverity := TRUE;
END_METHOD

METHOD SetEvent
VAR_INPUT
	EventId	  : UDINT;
	Trigger	  : POINTER TO BOOL;
	AutoReset : BOOL;
END_VAR

VAR
	pBool : POINTER TO BOOL;
END_VAR
IF CheckEventId(EventId) THEN
	IF Trigger <> 0 THEN
		SetEventTriggerInstance(EventId, Trigger);
	END_IF

	pBool  := GetEventAutoResetInstance(EventId);
	pBool^ := AutoReset;
END_IF
END_METHOD

METHOD SetEventReactions
VAR_INPUT
	Verbose	 : DINT := 0;
	Info	 : DINT := 1;
	Warning	 : DINT := 2;
	Error	 : DINT := 3;
	Critical : DINT := 4;
END_VAR
EventReactionVerbose  := Verbose;
EventReactionInfo	  := Info;
EventReactionWarning  := Warning;
EventReactionError	  := Error;
EventReactionCritical := Critical;
END_METHOD

METHOD PROTECTED CheckEventId : BOOL
VAR_INPUT
	EventId : UDINT;
END_VAR
CheckEventId := (EventID > 0) AND (EventId <= NumberOfEvents) AND (pEventBuffer <> 0);
END_METHOD

METHOD PROTECTED FindActiveSeverity
VAR
	i	   : UDINT;
	pEvent : POINTER TO FB_TcAlarm;
END_VAR
HighestActiveEventSeverity := Global.TcEventSeverity.Verbose;
FOR i := 1 TO NumberOfEvents DO
	pEvent := GetEventInstance(i);
	IF (pEvent <> 0) AND_THEN pEvent^.bRaised AND_THEN pEvent^.eSeverity > HighestActiveEventSeverity THEN
		HighestActiveEventSeverity := pEvent^.eSeverity;
	END_IF
END_FOR
END_METHOD

METHOD PROTECTED GetEventAutoResetInstance : POINTER TO BOOL
VAR_INPUT
	EventId : UDINT;
END_VAR

VAR
	ppEventAutoReset : POINTER TO POINTER TO BOOL;
END_VAR
IF CheckEventId(EventId) THEN
	ppEventAutoReset := pEventAutoResetBuffer + ((EventId - 1) * SIZEOF(PVOID));
	GetEventAutoResetInstance := ppEventAutoReset^;
ELSE
	GetEventAutoResetInstance := ADR(NullBool);
END_IF
END_METHOD

METHOD PROTECTED GetEventInstance : POINTER TO FB_TcAlarm
VAR_INPUT
	EventId : UDINT;
END_VAR

VAR
	ppEvent : POINTER TO POINTER TO FB_TcAlarm;
END_VAR
IF CheckEventId(EventId) THEN
	ppEvent			 := pEventBuffer + ((EventId - 1) * SIZEOF(PVOID));
	GetEventInstance := ppEvent^;
ELSE
	GetEventInstance := ADR(NullEvent);
END_IF
END_METHOD

METHOD PROTECTED GetEventTriggerInstance : POINTER TO BOOL
VAR_INPUT
	EventId : UDINT;
END_VAR

VAR
	ppEventTrigger : POINTER TO POINTER TO BOOL;
END_VAR
IF CheckEventId(EventId) THEN
	ppEventTrigger := pEventTriggerBuffer + ((EventId - 1) * SIZEOF(PVOID));
	GetEventTriggerInstance := ppEventTrigger^;
ELSE
	GetEventTriggerInstance := ADR(NullBool);
END_IF
END_METHOD

METHOD PROTECTED SetEventTriggerInstance
VAR_INPUT
	EventId : UDINT;
    Trigger : POINTER TO BOOL;
END_VAR

VAR
	ppEventTrigger : POINTER TO POINTER TO BOOL;
END_VAR
IF CheckEventId(EventId) THEN
	ppEventTrigger	:= pEventTriggerBuffer + ((EventId - 1) * SIZEOF(PVOID));
	ppEventTrigger^ := Trigger;
END_IF
END_METHOD

METHOD Reset
VAR
	i		 : UDINT;
	pEvent	 : POINTER TO FB_TcAlarm;
	pTrigger : POINTER TO BOOL;
END_VAR
FOR i := 1 TO NumberOfEvents DO
	pTrigger := GetEventTriggerInstance(i);
	pEvent	 := GetEventInstance(i);
	IF (pEvent <> 0) THEN
		IF (pTrigger <> 0) AND_THEN NOT pTrigger^ THEN
			pEvent^.Clear();
		END_IF

		IF (pTrigger = 0) THEN
			pEvent^.Clear();
		END_IF
	END_IF
END_FOR

HighestActiveEventSeverity := Global.TcEventSeverity.Verbose;
END_METHOD

METHOD PUBLIC Arguments : I_EventArguments
VAR_INPUT
	EventId : UDINT;
END_VAR

VAR
	pEvent : POINTER TO FB_TcAlarm;
END_VAR
IF CheckEventId(EventId) THEN
	pEvent := GetEventInstance(EventId);
	IF (pEvent <> 0) THEN
		TcEventClassArguments.Event := pEvent;
	ELSE
		TcEventClassArguments.Event := ADR(NullEvent);
	END_IF
ELSE
	TcEventClassArguments.Event := ADR(NullEvent);
END_IF

Arguments := TcEventClassArguments;
END_METHOD

METHOD CyclicLogic
VAR
	i	   : UDINT;
	pEvent : POINTER TO FB_TcAlarm;
	pTrigger  : POINTER TO BOOL;
    AutoReset : BOOL;
END_VAR
FOR i := 1 TO NumberOfEvents DO
	pTrigger := GetEventTriggerInstance(i);
	IF (pTrigger <> 0) THEN
		pEvent	  := GetEventInstance(i);
		AutoReset := GetEventAutoResetInstance(i)^;
		IF (pEvent <> 0) AND_THEN AutoReset AND NOT pTrigger^ THEN
			pEvent^.Clear();
			FindActiveSeverity();
		END_IF

		IF (pEvent <> 0) AND_THEN pTrigger^ THEN
			pEvent^.Raise(0);
			FindActiveSeverity();
		END_IF
	END_IF
END_FOR
END_METHOD

METHOD PUBLIC GenerateTcEvents
VAR_INPUT
	Name   : T_MaxString;
	pClass : PVOID; // ADR(TC_Events.XY) - TC Event Class in TypeSystem
	nSize  : UDINT; // SIZEOF(ST_XY) - TC Event Class in TypeSystem
END_VAR

VAR
	i				 : UDINT;
	pEventDef		 : POINTER TO TcEventEntry;
	pEvent			 : POINTER TO FB_TcAlarm;
	pBuffer			 : PVOID;
	ppBuffer		 : POINTER TO POINTER TO FB_TcAlarm;
	SourceInfo		 : FB_TcSourceInfo;
	pEventAutoReset	 : POINTER TO BOOL;
	ppEventAutoReset : POINTER TO POINTER TO BOOL;
END_VAR
NumberOfEvents		  := nSize / SIZEOF(TcEventEntry);
pEventBuffer		  := __NEW(PVOID, NumberOfEvents);
pEventTriggerBuffer	  := __NEW(PVOID, NumberOfEvents);
pEventAutoResetBuffer := __NEW(PVOID, NumberOfEvents);
pEventClass			  := pClass;
IF pEventBuffer <> 0 THEN
	SourceInfo.ResetToDefault();
	SourceInfo.sName := Name;
	FOR i := 1 TO NumberOfEvents DO
		pEvent	  := __NEW(FB_TcAlarm);
		ppBuffer  := pEventBuffer + ((i - 1) * SIZEOF(PVOID));
		ppBuffer^ := pEvent;
		pEventDef := pEventClass + ((i - 1) * SIZEOF(TcEventEntry));
		pEvent^.CreateEx2(pEventDef^, SourceInfo);

		//
		pEventAutoReset	  := __NEW(BOOL);
		ppEventAutoReset  := pEventAutoResetBuffer + ((i - 1) * SIZEOF(PVOID));
		ppEventAutoReset^ := pEventAutoReset;
	END_FOR
END_IF
END_METHOD

END_FUNCTION_BLOCK

// HMI/Interface/I_Button
INTERFACE I_Button EXTENDS I_Base

{attribute 'monitoring' := 'call'}
PROPERTY Active : BOOL
GET
END_GET
END_PROPERTY

{attribute 'monitoring' := 'call'}
PROPERTY Name : STRING
GET
END_GET
SET
END_SET
END_PROPERTY

PROPERTY Permissive : I_Permissive
GET
END_GET
END_PROPERTY

END_INTERFACE

// HMI/Interface/I_Permissive
INTERFACE I_Permissive EXTENDS I_Base

{attribute 'monitoring' := 'call'}
PROPERTY OK : BOOL
GET
END_GET
END_PROPERTY

METHOD Set
VAR_INPUT
	Index  : UDINT(0..9);
	Reason : STRING;
	Value  : BOOL;
END_VAR
END_METHOD

END_INTERFACE

// HMI/Interface/I_HmiFunction
INTERFACE I_HmiFunction EXTENDS I_Component

{attribute 'monitoring' := 'call'}
PROPERTY ControlType : STRING
GET
END_GET
SET
END_SET
END_PROPERTY

METHOD Disable
VAR_INPUT
END_VAR
END_METHOD

METHOD Enable
VAR_INPUT
END_VAR
END_METHOD

{attribute 'monitoring' := 'call'}
PROPERTY Enabled : BOOL
GET
END_GET
END_PROPERTY

{attribute 'monitoring' := 'call'}
PROPERTY InstancePath : STRING
GET
END_GET
END_PROPERTY

{attribute 'monitoring' := 'call'}
PROPERTY LinkObject : STRING
GET
END_GET
SET
END_SET
END_PROPERTY

END_INTERFACE

// HMI/Interface/I_StringCollection
INTERFACE I_StringCollection

METHOD AddString
VAR_INPUT
	StringToAdd : T_MaxString;
END_VAR
END_METHOD

METHOD Clear : BOOL
VAR_INPUT
END_VAR
END_METHOD

PROPERTY Entries : UDINT
GET
END_GET
END_PROPERTY

END_INTERFACE

// HMI/Button
FUNCTION_BLOCK Button IMPLEMENTS I_Button
VAR
	_Name		: STRING;
	_Active		: BOOL;
	_Permissive : PermissiveInterlock;
END_VAR

{attribute 'monitoring' := 'call'}
PROPERTY Active : BOOL
GET
Active := _Active;
END_GET
END_PROPERTY

{attribute 'monitoring' := 'call'}
PROPERTY Name : STRING
GET
Name := _Name;
END_GET
SET
_Name := Name;
END_SET
END_PROPERTY

PROPERTY Permissive : I_Permissive
GET
Permissive := _Permissive;
END_GET
END_PROPERTY

END_FUNCTION_BLOCK

// Permissive Interlock/PermissiveInterlock
FUNCTION_BLOCK PermissiveInterlock IMPLEMENTS I_Permissive
VAR
	_OK				 : BOOL				   := TRUE;
	Permissive		 : ARRAY[0..9] OF BOOL := [TRUE, TRUE, TRUE, TRUE, TRUE, TRUE, TRUE, TRUE, TRUE, TRUE];
	PermissiveReason : ARRAY[0..9] OF STRING;
END_VAR

METHOD PROTECTED Check : BOOL
VAR
	i : UDINT;
END_VAR
_OK := TRUE;
FOR i := 0 TO 9 DO
	IF NOT Permissive[i] THEN
		_OK := FALSE;
	END_IF
END_FOR
END_METHOD

{attribute 'monitoring' := 'call'}
PROPERTY OK : BOOL
GET
OK := _OK;
END_GET
END_PROPERTY

METHOD Set
VAR_INPUT
	Index  : UDINT(0..9);
	Reason : STRING;
	Value  : BOOL;
END_VAR
Permissive[Index]		:= Value;
PermissiveReason[Index] := Reason;
Check();
END_METHOD

END_FUNCTION_BLOCK

// HMI/HmiFunction
{attribute 'reflection'}
FUNCTION_BLOCK ABSTRACT HmiFunction EXTENDS CyclicComponent IMPLEMENTS I_HmiFunction
VAR
	{attribute 'instance-path'}
	{attribute 'noinit'}
	{attribute 'hide'}
	_InstancePath : STRING;
	{attribute 'hide'}
	_Enabled : BOOL := TRUE;
	{attribute 'hide'}
	_ControlType : STRING := 'Default';
	{attribute 'hide'}
	_LinkObject : STRING := 'DefaultFunction_HMI';
END_VAR

PROPERTY ABSTRACT ControlObject : I_Base
SET
END_SET
END_PROPERTY

{attribute 'monitoring' := 'call'}
PROPERTY ControlType : STRING
GET
ControlType := _ControlType;
END_GET
SET
_ControlType := ControlType;
END_SET
END_PROPERTY

METHOD CyclicLogic
END_METHOD

METHOD Disable
_Enabled := FALSE;
END_METHOD

METHOD Enable
_Enabled := TRUE;
END_METHOD

{attribute 'monitoring' := 'call'}
PROPERTY Enabled : BOOL
GET
Enabled := _Enabled;
END_GET
END_PROPERTY

{attribute 'monitoring' := 'call'}
PROPERTY InstancePath : STRING
GET
InstancePath := _InstancePath;
END_GET
END_PROPERTY

{attribute 'monitoring' := 'call'}
PROPERTY LinkObject : STRING
GET
LinkObject := _LinkObject;
END_GET
SET
_LinkObject := LinkObject;
END_SET
END_PROPERTY

END_FUNCTION_BLOCK

// Modes/PackMLModeControl
FUNCTION_BLOCK PackMLModeControl IMPLEMENTS I_Mode, I_Cyclic
VAR
	{attribute 'hide'}
	_CurrentMode : DINT;
	{attribute 'hide'}
	ModeManager	  : FB_PMLUnitModeManager;
	ModeCommand	  : DINT;
	_StateMachine : I_Statemachine;
END_VAR

METHOD ChangeMode
VAR_INPUT
	RequestedMode : DINT;
END_VAR
IF RequestedMode <= 0 OR RequestedMode > 31 THEN
	Trace.LogMessage('PackML Mode Controller', ' - Requested Mode is not valid 1..31');
	RETURN;
END_IF

ModeCommand := RequestedMode;
END_METHOD

{attribute 'monitoring' := 'call'}
PROPERTY CurrentMode : DINT
GET
CurrentMode := _CurrentMode;
END_GET
END_PROPERTY

METHOD CyclicLogic
VAR_INST
	LastModeCommand		: DINT;
	ModeChangeRequested : BOOL;
END_VAR
IF _CurrentMode = 0 THEN
	ModeChangeRequested := TRUE;
	ModeCommand			:= E_PMLProtectedUnitMode.Production;
	LastModeCommand		:= ModeCommand;
ELSIF ModeCommand <> LastModeCommand THEN
	ModeChangeRequested := TRUE;
	LastModeCommand		:= ModeCommand;
END_IF

IF ModeChangeRequested THEN
	{warning disable C0196}
	ModeManager(bExecute	 := TRUE,
				eModeCommand := ModeCommand,
				eState		 := _StateMachine.CurrentState,
				eModeStatus	 => _CurrentMode);

	IF ModeManager.bDone THEN
		ModeManager(bExecute := FALSE);
		ModeChangeRequested := FALSE;
	ELSIF ModeManager.bError THEN
		IF ModeManager.nErrorId = 1 THEN
			Trace.LogMessage('PackML Mode Controller', 'Requested mode is not defined or Mode change is disabled in this PackML state!');
		ELSE
			Trace.LogMessage('PackML Mode Controller', 'Mode change error, check PackML configuration!');
		END_IF

		ModeManager(bExecute := FALSE);
		_StateMachine.ChangeState(TO_UDINT(E_PMLCommand.Abort));
		ModeCommand			:= E_PMLProtectedUnitMode.Production;
		ModeChangeRequested := FALSE;
	END_IF
END_IF
END_METHOD

PROPERTY StateMachine : I_StateMachine
SET
_StateMachine := StateMachine;
END_SET
END_PROPERTY

END_FUNCTION_BLOCK

// Module PackML/PackMLModule
FUNCTION_BLOCK ABSTRACT PackMLModule EXTENDS Module IMPLEMENTS I_Module, I_ContainStatemachine
VAR
	_Statemachine : PackMLStatemachine_ModuleIntegrated('Statemachine');
	SequenceState : UDINT;
END_VAR

(*FB_Init is always available implicitly and it is used primarily for initialization.
The return value is not evaluated. For a specific influence, you can also declare the
methods explicitly and provide additional code there with the standard initialization
code. You can evaluate the return value.*)
METHOD FB_Init : BOOL
VAR_INPUT
	(* TRUE: the retain variables are initialized (reset warm / reset cold)*)
	bInitRetains	: BOOL;
	(* TRUE: the instance will be copied to the copy code afterward (online change)   *)
	bInCopyCode	: BOOL;
	Name	: T_MaxString;
END_VAR
_Statemachine.RegisterWithParent(THIS^);
END_METHOD

METHOD Aborted : BOOL;
Aborted := TRUE;
END_METHOD

METHOD Aborting : BOOL
Aborting := TRUE;
END_METHOD

METHOD Clearing : BOOL
Clearing := TRUE;
END_METHOD

METHOD Completed : BOOL
Completed := TRUE;
END_METHOD

METHOD Completing : BOOL
Completing := TRUE;
END_METHOD

METHOD Execute : BOOL
Execute := TRUE;
END_METHOD

METHOD Held : BOOL
Held := TRUE;
END_METHOD

METHOD Holding : BOOL
Holding := TRUE;
END_METHOD

METHOD Idle : BOOL
Idle := TRUE;
END_METHOD

METHOD Resetting : BOOL
Resetting := TRUE;
END_METHOD

METHOD Starting : BOOL
Starting := TRUE;
END_METHOD

METHOD Stopped : BOOL
Stopped := TRUE;
END_METHOD

METHOD Stopping : BOOL
Stopping := TRUE;
END_METHOD

METHOD Suspended : BOOL
Suspended := TRUE;
END_METHOD

METHOD Suspending : BOOL
Suspending := TRUE;
END_METHOD

METHOD Unholding : BOOL
Unholding := TRUE;
END_METHOD

METHOD Unsuspending : BOOL
Unsuspending := TRUE;
END_METHOD

METHOD CyclicLogic
StateSelect();
SUPER^.CyclicLogic();
END_METHOD

PROPERTY Statemachine : I_Statemachine
GET
Statemachine := _Statemachine;
END_GET
END_PROPERTY

METHOD PRIVATE StateSelect
VAR_INST
	ClearingTon : TON;
	LastState	: DINT;
END_VAR
IF LastState <> _Statemachine.CurrentState THEN
	SequenceState := 0;
	LastState	  := _Statemachine.CurrentState;
END_IF

CASE _Statemachine.CurrentState OF
	E_PMLState.Undefined:
		;

	E_PMLState.Clearing:
		ClearingTon(IN := TRUE, PT := CoreParameter.ClearingTimeout);
		IF Clearing() THEN
			ClearingTon(IN := FALSE);
			_Statemachine.StateComplete();
		END_IF

		IF ClearingTon.Q THEN
			ClearingTon(IN := FALSE);
			Trace.LogMessage('Clearing Timeout exeeded! - ', _Name);
			_Statemachine.ChangeState(E_PMLCommand.Abort);
		END_IF

	E_PMLState.Stopped:
		Stopped();

	E_PMLState.Starting:
		IF Starting() THEN
			_Statemachine.StateComplete();
		END_IF

	E_PMLState.Idle:
		Idle();

	E_PMLState.Suspended:
		Suspended();

	E_PMLState.Execute:
		Execute();

	E_PMLState.Stopping:
		IF Stopping() THEN
			_Statemachine.StateComplete();
		END_IF

	E_PMLState.Aborting:
		IF Aborting() THEN
			_Statemachine.StateComplete();
		END_IF

	E_PMLState.Aborted:
		Aborted();

	E_PMLState.Holding:
		IF Holding() THEN
			_Statemachine.StateComplete();
		END_IF

	E_PMLState.Held:
		Held();

	E_PMLState.Unholding:
		IF Unholding() THEN
			_Statemachine.StateComplete();
		END_IF

	E_PMLState.Suspending:
		IF Suspending() THEN
			_Statemachine.StateComplete();
		END_IF

	E_PMLState.Unsuspending:
		IF Unsuspending() THEN
			_Statemachine.StateComplete();
		END_IF

	E_PMLState.Resetting:
		IF Resetting() THEN
			_Statemachine.StateComplete();
		END_IF

	E_PMLState.Completing:
		IF Completing() THEN
			_Statemachine.StateComplete();
		END_IF

	E_PMLState.Completed:
		Completed();
END_CASE
END_METHOD

END_FUNCTION_BLOCK

// Statemachine/Interface/I_ContainStatemachine
INTERFACE I_ContainStatemachine EXTENDS I_Base

PROPERTY Statemachine : I_Statemachine
GET
END_GET
END_PROPERTY

END_INTERFACE

// Statemachine/PackML/PackMLStatemachine_ModuleIntegrated
FUNCTION_BLOCK PackMLStatemachine_ModuleIntegrated EXTENDS CyclicComponent IMPLEMENTS I_StateMachine
VAR
	StateMachine   : FB_PMLStateMachine;
	StateCommand   : E_PMLCommand;
	_CurrentState  : E_PMLState;
	ModeController : PackMLModeControl := (StateMachine := THIS^);
END_VAR

PROPERTY Mode : I_Mode
GET
Mode := ModeController;
END_GET
SET
// Fix defined in PackML
END_SET
END_PROPERTY

METHOD ChangeState
VAR_INPUT
	StateCommand : DINT;
END_VAR
IF StateCommand <= 0 OR StateCommand > 17 THEN
	Trace.LogMessage('PackML Statemachine ChangeState()', 'StateId is not a PackML State');
END_IF

{warning disable C0196}
THIS^.StateCommand := StateCommand;
END_METHOD

{attribute 'monitoring' := 'call'}
PROPERTY CurrentState : DINT
GET
CurrentState := _CurrentState;
END_GET
END_PROPERTY

METHOD CyclicLogic
VAR_INST
	ClearingTon : TON;
END_VAR
ModeController.CyclicLogic();
IF _CurrentState = E_PMLState.Undefined AND Mode.CurrentMode <> 0 THEN
	StateCommand := E_PMLCommand.Abort;
END_IF

StateMachine(eMode			  := TO_DINT(Mode.CurrentMode),
			 eCommand		  := StateCommand,
			 stSubUnitInfoRef :=,
			 stOptions		  :=,
			 eState			  => _CurrentState,
			 sState			  =>,
			 bError			  =>,
			 nErrorID		  =>);

CASE _CurrentState OF
	E_PMLState.Clearing:
		ClearingTon(IN := TRUE, PT := CoreParameter.ClearingTimeout);
		IF ClearingTon.Q THEN
			ClearingTon(IN := FALSE);
			Trace.LogMessage('Clearing Timeout exeeded!', 'CoreParameter.ClearingTimeout');
			StateCommand := E_PMLCommand.Abort;
		END_IF

ELSE
	ClearingTon(IN := FALSE);
END_CASE
END_METHOD

METHOD StateComplete
StateMachine.M_StateComplete();
END_METHOD

{attribute 'hide'} 
PROPERTY States : I_StateList
GET
States := 0;
END_GET
END_PROPERTY

END_FUNCTION_BLOCK

// Project Information/F_GetCompany
// This function has been automatically generated from the project information.
{attribute 'signature_flag' := '1073741824'}
{attribute 'TcGenerated'}
{attribute 'no-analysis'}
FUNCTION F_GetCompany : WSTRING
VAR_INPUT
	
END_VAR

F_GetCompany := "Beckhoff Automation LLC";

END_FUNCTION

// Project Information/F_GetTitle
// This function has been automatically generated from the project information.
{attribute 'signature_flag' := '1073741824'}
{attribute 'TcGenerated'}
{attribute 'no-analysis'}
FUNCTION F_GetTitle : WSTRING
VAR_INPUT
	
END_VAR

F_GetTitle := "Core";

END_FUNCTION

// Project Information/F_GetVersion
// This function has been automatically generated from the project information.
{attribute 'signature_flag' := '1073741824'}
{attribute 'TcGenerated'}
{attribute 'no-analysis'}
FUNCTION F_GetVersion : ST_LibVersion
VAR_INPUT
	
END_VAR

F_GetVersion.iMajor := 1;
F_GetVersion.iMinor := 3;
F_GetVersion.iBuild := 3;
F_GetVersion.iRevision := 0;
F_GetVersion.sVersion := '1.3.3';
F_GetVersion.nFlags := 0;

END_FUNCTION

// Statemachine/Generic/NextMinorStep
FUNCTION NextMinorStep : UDINT
VAR_IN_OUT
	StateVar : UDINT;
END_VAR

NextMinorStep := StateVar := StateVar + 1;

END_FUNCTION

// Statemachine/Generic/NextStep
FUNCTION NextStep : UDINT
VAR_IN_OUT
	StateVar : UDINT;
END_VAR

NextStep := StateVar := ((StateVar / 10) * 10) + 10;

END_FUNCTION

// Statemachine/Generic/SetStep
FUNCTION SetStep : UDINT
VAR_IN_OUT
	StateVar : UDINT;
END_VAR

VAR_INPUT
	Step : UDINT;
END_VAR

SetStep := StateVar := Step;

END_FUNCTION

// Statemachine/Generic/Statemachine_HMI
FUNCTION_BLOCK Statemachine_HMI EXTENDS HmiFunction
VAR
	Statemachine : I_Statemachine;
	{ attribute 'TcHmiSymbol.AddSymbol' }
	{ attribute 'TcHmiSymbol.AddSymbol.UserGroups' := '__SystemAdministrators,Admin' }
	Statemachine_HMI : ST_Statemachine_HMI;
END_VAR

PROPERTY ControlObject : I_Base
SET
__QueryInterface(ControlObject,Statemachine);
END_SET
END_PROPERTY

METHOD CyclicLogic
VAR_INST
	LastModeChangeCommand  : DINT;
	LastStateChangeCommand : DINT;
END_VAR
Statemachine_HMI.Name		  := Statemachine.Name;
Statemachine_HMI.CurrentState := Statemachine.CurrentState;
Statemachine_HMI.CurrentMode  := Statemachine.Mode.CurrentMode;
Statemachine_HMI.HmiEnabled	  := Enabled;
IF Enabled THEN
	IF Statemachine_HMI.ModeChangeCommand <> 0 THEN
		Statemachine.Mode.ChangeMode(Statemachine_HMI.ModeChangeCommand);
		LastModeChangeCommand			   := Statemachine_HMI.ModeChangeCommand;
		Statemachine_HMI.ModeChangeCommand := 0;
	END_IF

	{warning disable C0196}
	IF Statemachine_HMI.StateChangeCommand <> 0 THEN
		Statemachine.ChangeState(TO_UDINT(Statemachine_HMI.StateChangeCommand));
		{warning disable C0195}
		LastStateChangeCommand				:= Statemachine_HMI.StateChangeCommand;
		Statemachine_HMI.StateChangeCommand := 0;
	END_IF
ELSE
	Statemachine_HMI.StateChangeCommand := 0;
	Statemachine_HMI.ModeChangeCommand	:= 0;
END_IF
END_METHOD

(*FB_Init is always available implicitly and it is used primarily for initialization.
The return value is not evaluated. For a specific influence, you can also declare the
methods explicitly and provide additional code there with the standard initialization
code. You can evaluate the return value.*)
METHOD FB_Init : BOOL
VAR_INPUT
	(* TRUE: the retain variables are initialized (reset warm / reset cold)*)
	bInitRetains : BOOL;

	(* TRUE: the instance will be copied to the copy code afterward (online change)   *)
	bInCopyCode	 : BOOL;
	Name		 : T_MaxString;
	Statemachine : I_Statemachine;
END_VAR
THIS^.Statemachine := Statemachine;
ControlType		   := 'Statemachine';
LinkObject		   := 'Statemachine_HMI';
END_METHOD

END_FUNCTION_BLOCK

// Statemachine/PackML/NextAvailablePackMLCommands
FUNCTION_BLOCK NextAvailablePackMLCommands
VAR
	NextAvailableCommands : ARRAY[0..MAX_AVAILABLE_COMMANDS] OF E_PMLCommand;
	i					  : UDINT;
END_VAR

VAR CONSTANT
	MAX_AVAILABLE_COMMANDS : UDINT := 9;
END_VAR

METHOD PUBLIC GetCommands : ARRAY[0..MAX_AVAILABLE_COMMANDS] OF E_PMLCommand
VAR_INPUT
	CurrentMode	 : DINT(0..31);
	CurrentState : E_PMLState;
END_VAR

VAR
	ModeConfiguration : Tc3_PackML_V3.ST_PMLUnitModeConfiguration;
END_VAR
FOR i := 1 TO MAX_AVAILABLE_COMMANDS DO
	NextAvailableCommands[i] := E_PMLCommand.Undefined;
END_FOR

i				  := 0;
ModeConfiguration := Tc3_PackML_V3.GlobalVariables.stPMLUnitModeConfiguration[CurrentMode];
// Generate next possible Commands
CASE CurrentState OF
	E_PMLState.Undefined:
		;

	E_PMLState.Aborting:
		;

	E_PMLState.Aborted:
		NextAvailableCommands[i] := E_PMLCommand.Clear;

	E_PMLState.Clearing:
		;

	E_PMLState.Stopping:
		NextAvailableCommands[i] := E_PMLCommand.Abort;

	E_PMLState.Stopped:
		NextAvailableCommands[i] := E_PMLCommand.Abort;
		i						 := i + 1;
		IF NOT ModeConfiguration.aStateDisabled[E_PMLState.Resetting] AND NOT ModeConfiguration.aStateDisabled[E_PMLState.Idle] THEN
			NextAvailableCommands[i] := E_PMLCommand.Reset;
		ELSE
			NextAvailableCommands[i] := E_PMLCommand.Start;
		END_IF

	E_PMLState.Resetting:
		NextAvailableCommands[i] := E_PMLCommand.Abort;
		i						 := i + 1;
		NextAvailableCommands[i] := E_PMLCommand.Stop;

	E_PMLState.Idle:
		NextAvailableCommands[i] := E_PMLCommand.Abort;
		i						 := i + 1;
		NextAvailableCommands[i] := E_PMLCommand.Stop;
		i						 := i + 1;
		NextAvailableCommands[i] := E_PMLCommand.Start;

	E_PMLState.Starting:
		NextAvailableCommands[i] := E_PMLCommand.Abort;
		i						 := i + 1;
		NextAvailableCommands[i] := E_PMLCommand.Stop;

	E_PMLState.Execute:
		NextAvailableCommands[i] := E_PMLCommand.Abort;
		i						 := i + 1;
		NextAvailableCommands[i] := E_PMLCommand.Stop;
		i						 := i + 1;
		IF (NOT ModeConfiguration.aStateDisabled[E_PMLState.Held] AND NOT ModeConfiguration.aStateDisabled[E_PMLState.Holding]) OR (NOT ModeConfiguration.aStateDisabled[E_PMLState.Held] AND NOT ModeConfiguration.aStateDisabled[E_PMLState.Unholding]) THEN
			NextAvailableCommands[i] := E_PMLCommand.Hold;
			i						 := i + 1;
		END_IF

		IF (NOT ModeConfiguration.aStateDisabled[E_PMLState.Suspended] AND NOT ModeConfiguration.aStateDisabled[E_PMLState.Suspending]) OR (NOT ModeConfiguration.aStateDisabled[E_PMLState.Suspended] AND NOT ModeConfiguration.aStateDisabled[E_PMLState.Unsuspending]) THEN
			NextAvailableCommands[i] := E_PMLCommand.Suspend;
			i						 := i + 1;
		END_IF

		IF NOT ModeConfiguration.aStateDisabled[E_PMLState.Completed] AND NOT ModeConfiguration.aStateDisabled[E_PMLState.Completing] THEN
			NextAvailableCommands[i] := E_PMLCommand.Complete;
			i						 := i + 1;
		ELSIF NOT ModeConfiguration.aStateDisabled[E_PMLState.Resetting] THEN
			NextAvailableCommands[i] := E_PMLCommand.Reset;
			i						 := i + 1;
		END_IF

	E_PMLState.Completing:
		NextAvailableCommands[i] := E_PMLCommand.Abort;
		i						 := i + 1;
		NextAvailableCommands[i] := E_PMLCommand.Stop;

	E_PMLState.Completed:
		NextAvailableCommands[i] := E_PMLCommand.Abort;
		i						 := i + 1;
		NextAvailableCommands[i] := E_PMLCommand.Stop;
		i						 := i + 1;
		IF NOT ModeConfiguration.aStateDisabled[E_PMLState.Resetting] AND NOT ModeConfiguration.aStateDisabled[E_PMLState.Idle] THEN
			NextAvailableCommands[i] := E_PMLCommand.Reset;
		ELSE
			NextAvailableCommands[i] := E_PMLCommand.Start;
		END_IF

	E_PMLState.Holding:
		NextAvailableCommands[i] := E_PMLCommand.Abort;
		i						 := i + 1;
		NextAvailableCommands[i] := E_PMLCommand.Stop;

	E_PMLState.Held:
		NextAvailableCommands[i] := E_PMLCommand.Abort;
		i						 := i + 1;
		NextAvailableCommands[i] := E_PMLCommand.Stop;
		i						 := i + 1;
		NextAvailableCommands[i] := E_PMLCommand.Unhold;

	E_PMLState.Unholding:
		NextAvailableCommands[i] := E_PMLCommand.Abort;
		i						 := i + 1;
		NextAvailableCommands[i] := E_PMLCommand.Stop;

	E_PMLState.Suspending:
		NextAvailableCommands[i] := E_PMLCommand.Abort;
		i						 := i + 1;
		NextAvailableCommands[i] := E_PMLCommand.Stop;

	E_PMLState.Suspended:
		NextAvailableCommands[i] := E_PMLCommand.Abort;
		i						 := i + 1;
		NextAvailableCommands[i] := E_PMLCommand.Stop;
		i						 := i + 1;
		NextAvailableCommands[i] := E_PMLCommand.Unsuspend;

	E_PMLState.Unsuspending:
		NextAvailableCommands[i] := E_PMLCommand.Abort;
		i						 := i + 1;
		NextAvailableCommands[i] := E_PMLCommand.Stop;
END_CASE

GetCommands := NextAvailableCommands;
END_METHOD

END_FUNCTION_BLOCK

// Statemachine/PackML/PackMLStatemachine
FUNCTION_BLOCK PackMLStatemachine EXTENDS CyclicComponent IMPLEMENTS I_StateMachine
VAR
	StateList	   : StateList<17>;
	StateMachine   : FB_PMLStateMachine;
	StateCommand   : E_PMLCommand;
	_CurrentState  : E_PMLState;
	ModeController : PackMLModeControl := (StateMachine := THIS^);
END_VAR

PROPERTY Mode : I_Mode
GET
Mode := ModeController;
END_GET
SET
// Fix defined in PackML
END_SET
END_PROPERTY

METHOD PROTECTED CallState : BOOL
VAR_INPUT
	StateIndex : E_PMLState;
END_VAR

VAR
	State : I_State;
	i	  : DINT;
END_VAR
State := StateList.GetStateAtIndex(StateIndex);
IF State <> 0 THEN
	CallState := State.Executing();
ELSE
	CallState := TRUE;
END_IF

FOR i := 0 TO StateList.NumberOfStates DO
	State := StateList.GetStateAtIndex(i);
	IF State <> 0 AND i <> StateIndex THEN
		State.Inactive();
	END_IF
END_FOR
END_METHOD

METHOD ChangeState
VAR_INPUT
	StateCommand : DINT;
END_VAR
IF StateCommand <= 0 OR StateCommand > 17 THEN
	Trace.LogMessage('PackML Statemachine ChangeState()', 'StateId is not a PackML State');
END_IF

{warning disable C0196}
THIS^.StateCommand := StateCommand;
END_METHOD

{attribute 'monitoring' := 'call'}
PROPERTY CurrentState : DINT
GET
CurrentState := _CurrentState;
END_GET
END_PROPERTY

PROPERTY States : I_StateList
GET
States := StateList;
END_GET
END_PROPERTY

